(* IEC 61131-3 sources: SmartHomeNew/ (part 5) *)

(* ---- FB_Heating_Adaptive_Target.st ---- *)
// ==============================================================================
// Adaptive target calculation for heating supply temperature
// ==============================================================================
FUNCTION_BLOCK FB_Heating_Adaptive_Target
VAR_INPUT
    VI_Base_Target_Supply_Temp : REAL;
    VI_Global_Target_Temperature : REAL;
END_VAR

VAR_IN_OUT
    VI_Zone_Configs : ARRAY[1..GVL_CONSTANTS.C_MAX_HEATING_CIRCUITS] OF ST_FloorHeating_Circuit_Config;
    VI_Floor_Temps : ARRAY[1..GVL_CONSTANTS.C_MAX_HEATING_CIRCUITS] OF REAL;
    VI_Room_Temps : ARRAY[1..GVL_CONSTANTS.C_MAX_ZONES] OF REAL;
END_VAR

VAR_OUTPUT
    VO_Target_Supply_Temp : REAL;
    VO_Adaptive_Correction : REAL;
    VO_Adaptive_Effective_Delta : REAL;
    VO_Adaptive_Max_Delta : REAL;
END_VAR

VAR
    L_Adaptive_Zone_i : INT;
    L_Zone_Index : INT;
    L_Adaptive_Delta : REAL;
    L_Adaptive_Weighted_Sum : REAL;
    L_Adaptive_Weight_Total : REAL;
    L_Adaptive_Weight : REAL;
END_VAR

VO_Target_Supply_Temp := VI_Base_Target_Supply_Temp;
VO_Adaptive_Max_Delta := 0.0;
L_Adaptive_Weighted_Sum := 0.0;
L_Adaptive_Weight_Total := 0.0;
VO_Adaptive_Effective_Delta := 0.0;
VO_Adaptive_Correction := 0.0;

IF VI_Global_Target_Temperature > 0.0 THEN
    VO_Target_Supply_Temp := VI_Global_Target_Temperature;
END_IF;

FOR L_Adaptive_Zone_i := 1 TO GVL_CONSTANTS.C_MAX_HEATING_CIRCUITS DO
    L_Zone_Index := VI_Zone_Configs[L_Adaptive_Zone_i].zone;

    IF (L_Zone_Index >= 1) AND (L_Zone_Index <= GVL_CONSTANTS.C_MAX_ZONES) THEN
        CASE VI_Zone_Configs[L_Adaptive_Zone_i].control_type OF
            0:
                L_Adaptive_Delta :=
                    VI_Zone_Configs[L_Adaptive_Zone_i].design_temp -
                    VI_Floor_Temps[L_Adaptive_Zone_i];
                L_Adaptive_Weight := 0.6;
            1, 2:
                L_Adaptive_Delta :=
                    VI_Zone_Configs[L_Adaptive_Zone_i].design_temp -
                    VI_Room_Temps[L_Zone_Index];
                L_Adaptive_Weight := 1.0;
            ELSE
                L_Adaptive_Delta :=
                    VI_Zone_Configs[L_Adaptive_Zone_i].design_temp -
                    VI_Room_Temps[L_Zone_Index];
                L_Adaptive_Weight := 0.8;
        END_CASE;

        IF L_Zone_Index <= 4 THEN
            L_Adaptive_Weight := L_Adaptive_Weight * 1.2;
        ELSIF L_Zone_Index >= 9 THEN
            L_Adaptive_Weight := L_Adaptive_Weight * 0.7;
        END_IF;

        IF L_Adaptive_Weight > 2.0 THEN
            L_Adaptive_Weight := 2.0;
        ELSIF L_Adaptive_Weight < 0.2 THEN
            L_Adaptive_Weight := 0.2;
        END_IF;

        IF L_Adaptive_Delta > VO_Adaptive_Max_Delta THEN
            VO_Adaptive_Max_Delta := L_Adaptive_Delta;
        END_IF;

        L_Adaptive_Weighted_Sum := L_Adaptive_Weighted_Sum + (L_Adaptive_Delta * L_Adaptive_Weight);
        L_Adaptive_Weight_Total := L_Adaptive_Weight_Total + L_Adaptive_Weight;
    END_IF;
END_FOR;

IF L_Adaptive_Weight_Total > 0.0 THEN
    VO_Adaptive_Effective_Delta := L_Adaptive_Weighted_Sum / L_Adaptive_Weight_Total;
END_IF;

IF VO_Adaptive_Effective_Delta > 1.5 THEN
    VO_Adaptive_Correction := 2.0;
ELSIF VO_Adaptive_Effective_Delta > 0.7 THEN
    VO_Adaptive_Correction := 1.0;
ELSIF VO_Adaptive_Effective_Delta < -1.5 THEN
    VO_Adaptive_Correction := -2.0;
ELSIF VO_Adaptive_Effective_Delta < -0.7 THEN
    VO_Adaptive_Correction := -1.0;
ELSE
    VO_Adaptive_Correction := 0.0;
END_IF;

IF VO_Adaptive_Max_Delta > 2.5 AND VO_Adaptive_Correction < 2.0 THEN
    VO_Adaptive_Correction := 2.0;
END_IF;

VO_Target_Supply_Temp := VO_Target_Supply_Temp + VO_Adaptive_Correction;

IF VO_Target_Supply_Temp < 20.0 THEN
    VO_Target_Supply_Temp := 20.0;
ELSIF VO_Target_Supply_Temp > 45.0 THEN
    VO_Target_Supply_Temp := 45.0;
END_IF;

// >>> BULK_SYNC_ANCHOR: FB_Heating_Adaptive_Target <<<

(* ---- FB_Heating_Allocation_Filter.st ---- *)
// ==============================================================================
// Heating allocation filter
// Bounded policy filter between demand map and manifold control.
//
// Purpose:
// - preserve current runtime ownership;
// - avoid reconnecting legacy orchestration wrappers;
// - provide a safe insertion point for selective thermal allocation logic;
// - keep default behavior transparent when disabled.
//
// This FB does NOT own:
// - heating orchestration;
// - boiler control;
// - valve control;
// - pump control;
// - safety state;
// - output projection.
//
// Migration source:
// - useful bounded logic from FB_Heating_Thermal_Allocation;
// - useful bounded logic from FB_Heating_Decision_Context.
//
// Explicitly not migrated:
// - FB_Heating_Orchestration wrapper;
// - FB_Heating_Execution_Core wrapper;
// - FB_Heating_Override_Layer hard output authority.
// ==============================================================================
FUNCTION_BLOCK FB_Heating_Allocation_Filter
VAR_INPUT
    // Master switch for any filtering.
    // FALSE means strict passthrough: output demand equals input demand.
    VI_Enable : BOOL;

    // Enables optional priority/budget allocation.
    // FALSE means only safe availability filtering may run when VI_Enable is TRUE.
    VI_Enable_Policy_Allocation : BOOL := FALSE;

    // Current demand from FB_Heating_Demand_Map.
    VI_Manifold_Demand_Map : ARRAY[1..GVL_CONSTANTS.C_MAX_MANIFOLDS] OF BOOL;

    // Availability must come from current active owners / diagnostics.
    // TRUE means the manifold is allowed to receive demand.
    VI_Manifold_Available : ARRAY[1..GVL_CONSTANTS.C_MAX_MANIFOLDS] OF BOOL;

    // Optional policy inputs staged for future activation.
    // They intentionally stay outside existing DUT/GVL contract for now.
    VI_Manifold_Base_Priority : ARRAY[1..GVL_CONSTANTS.C_MAX_MANIFOLDS] OF INT;
    VI_Manifold_Thermal_Weight : ARRAY[1..GVL_CONSTANTS.C_MAX_MANIFOLDS] OF REAL;
    VI_Max_Thermal_Budget : REAL := REAL#0.0;
END_VAR
VAR_OUTPUT
    // Demand forwarded to FB_Heating_Manifold_Control.
    VO_Manifold_Demand_Filtered : ARRAY[1..GVL_CONSTANTS.C_MAX_MANIFOLDS] OF BOOL;

    // TRUE when at least one demanded manifold was blocked by availability or policy.
    VO_Allocation_Degraded : BOOL;

    // Diagnostic outputs for later observation/HMI integration.
    VO_Manifold_Allowed : ARRAY[1..GVL_CONSTANTS.C_MAX_MANIFOLDS] OF BOOL;
    VO_Manifold_Priority_Effective : ARRAY[1..GVL_CONSTANTS.C_MAX_MANIFOLDS] OF INT;
    VO_Thermal_Budget_Used : REAL;
END_VAR
VAR
    L_i : INT;
    L_CurrentPriority : INT;
    L_MaxPriority : INT;
    L_Used : REAL;
    L_Weight : REAL;
END_VAR

// ======================================================
// DEFAULT / TRANSPARENT MODE
// ======================================================
VO_Allocation_Degraded := FALSE;
VO_Thermal_Budget_Used := REAL#0.0;

FOR L_i := 1 TO GVL_CONSTANTS.C_MAX_MANIFOLDS DO
    VO_Manifold_Demand_Filtered[L_i] := VI_Manifold_Demand_Map[L_i];
    VO_Manifold_Allowed[L_i] := TRUE;
    VO_Manifold_Priority_Effective[L_i] := VI_Manifold_Base_Priority[L_i];
END_FOR;

IF NOT VI_Enable THEN
    RETURN;
END_IF;

// ======================================================
// SAFE AVAILABILITY FILTER
// ======================================================
FOR L_i := 1 TO GVL_CONSTANTS.C_MAX_MANIFOLDS DO
    VO_Manifold_Allowed[L_i] := VI_Manifold_Available[L_i];

    IF VI_Manifold_Demand_Map[L_i] AND NOT VO_Manifold_Allowed[L_i] THEN
        VO_Manifold_Demand_Filtered[L_i] := FALSE;
        VO_Allocation_Degraded := TRUE;
    END_IF;
END_FOR;

// ======================================================
// OPTIONAL POLICY / THERMAL BUDGET ALLOCATION
// ======================================================
IF NOT VI_Enable_Policy_Allocation THEN
    RETURN;
END_IF;

// Invalid or unset budget means do not apply budget shedding.
IF VI_Max_Thermal_Budget <= REAL#0.0 THEN
    RETURN;
END_IF;

// Clear filtered demand before rebuilding it by priority and budget.
FOR L_i := 1 TO GVL_CONSTANTS.C_MAX_MANIFOLDS DO
    VO_Manifold_Demand_Filtered[L_i] := FALSE;
END_FOR;

// Find max priority among demanded and allowed manifolds.
L_MaxPriority := 0;
FOR L_i := 1 TO GVL_CONSTANTS.C_MAX_MANIFOLDS DO
    IF VI_Manifold_Demand_Map[L_i] AND VO_Manifold_Allowed[L_i] THEN
        IF VO_Manifold_Priority_Effective[L_i] > L_MaxPriority THEN
            L_MaxPriority := VO_Manifold_Priority_Effective[L_i];
        END_IF;
    END_IF;
END_FOR;

L_Used := REAL#0.0;

FOR L_CurrentPriority := L_MaxPriority TO 0 BY -1 DO
    FOR L_i := 1 TO GVL_CONSTANTS.C_MAX_MANIFOLDS DO
        IF VI_Manifold_Demand_Map[L_i]
           AND VO_Manifold_Allowed[L_i]
           AND (VO_Manifold_Priority_Effective[L_i] = L_CurrentPriority) THEN

            L_Weight := VI_Manifold_Thermal_Weight[L_i];
            IF L_Weight <= REAL#0.0 THEN
                L_Weight := REAL#1.0;
            END_IF;

            IF (L_Used + L_Weight) <= VI_Max_Thermal_Budget THEN
                VO_Manifold_Demand_Filtered[L_i] := TRUE;
                L_Used := L_Used + L_Weight;
            ELSE
                VO_Allocation_Degraded := TRUE;
            END_IF;
        END_IF;
    END_FOR;
END_FOR;

VO_Thermal_Budget_Used := L_Used;

END_FUNCTION_BLOCK
// >>> BULK_SYNC_ANCHOR: FB_Heating_Allocation_Filter <<<

(* ---- FB_Heating_Boiler_Control.st ---- *)
// ==============================================================================
// Heating boiler control helper
// ==============================================================================
FUNCTION_BLOCK FB_Heating_Boiler_Control
VAR_INPUT
    VI_System_Time_MS : UDINT;
    VI_IsActivePLC : BOOL;
    VI_DHW_Heating_Demand : BOOL;
    VI_DHW_Target_Temp : REAL;
    VI_Target_Supply_Temp : REAL;
    VI_Freeze_Mode_Active : BOOL;
    VI_Policy_Degraded : BOOL;
    VI_Manifold_Pumps : ARRAY[1..GVL_CONSTANTS.C_MAX_MANIFOLDS] OF BOOL;
    VI_Manifold_Valves : ARRAY[1..GVL_CONSTANTS.C_MAX_MANIFOLDS] OF REAL;
    VI_Boiler_Flame_Status : ARRAY[1..GVL_CONSTANTS.C_MAX_BOILERS] OF BOOL;
    VI_Boiler_Error_Status : ARRAY[1..GVL_CONSTANTS.C_MAX_BOILERS] OF BOOL;
    VI_Boiler_OT_Online : ARRAY[1..GVL_CONSTANTS.C_MAX_BOILERS] OF BOOL;
END_VAR
VAR_IN_OUT
    VI_Boiler_Modulation : ARRAY[1..GVL_CONSTANTS.C_MAX_BOILERS] OF REAL;
END_VAR
VAR_OUTPUT
    VO_Boiler_OT_Enable : ARRAY[1..GVL_CONSTANTS.C_MAX_BOILERS] OF BOOL;
    VO_Boiler_OT_Setpoint : ARRAY[1..GVL_CONSTANTS.C_MAX_BOILERS] OF REAL;
    VO_Boiler_Status : ARRAY[1..GVL_CONSTANTS.C_MAX_BOILERS] OF ST_Boiler_Status;
    VO_Any_Subsystem_Degraded : BOOL;
    VO_Lead_Boiler : BYTE;
    VO_Demand_Power : REAL;
END_VAR
VAR
    L_i : INT;
    L_Delta_MS : UDINT;
    L_Last_Scan_Time : UDINT;
    L_Scan_Time_Init : BOOL := FALSE;
    L_Boiler_Request_Enable : ARRAY[1..GVL_CONSTANTS.C_MAX_BOILERS] OF BOOL;
    L_Boiler_Request_Setpoint : ARRAY[1..GVL_CONSTANTS.C_MAX_BOILERS] OF REAL;
    L_Boiler_OT_Command_Valid : ARRAY[1..GVL_CONSTANTS.C_MAX_BOILERS] OF BOOL;
    L_Transport_Degraded : BOOL;
    L_Available_Count : UINT;
    L_Active_Count : UINT;
    L_Any_Transport_Degraded : BOOL;
    L_Any_Ignition_Timeout : BOOL;
    L_Any_Flame : BOOL;
    L_Empty_Boiler_Status : ST_Boiler_Status;
    L_Boiler_Life : ARRAY[1..GVL_CONSTANTS.C_MAX_BOILERS] OF FB_Lifetime_Predictor;
    fbBoilerCascade : FB_Boiler_Cascade_Manager;
    fbBoilerOpenTherm : FB_Boiler_OpenTherm_Interface;
END_VAR

VO_Any_Subsystem_Degraded := FALSE;
VO_Lead_Boiler := 0;
VO_Demand_Power := 0.0;

L_Available_Count := 0;
L_Active_Count := 0;
L_Any_Transport_Degraded := FALSE;
L_Any_Ignition_Timeout := FALSE;
L_Any_Flame := FALSE;

FOR L_i := 1 TO GVL_CONSTANTS.C_MAX_BOILERS DO
    L_Boiler_Request_Enable[L_i] := FALSE;
    L_Boiler_Request_Setpoint[L_i] := 0.0;
    L_Boiler_OT_Command_Valid[L_i] := FALSE;
    VO_Boiler_OT_Enable[L_i] := FALSE;
    VO_Boiler_OT_Setpoint[L_i] := 0.0;
    VO_Boiler_Status[L_i] := L_Empty_Boiler_Status;
END_FOR;

FOR L_i := 1 TO GVL_CONSTANTS.C_MAX_MANIFOLDS DO
    IF VI_Manifold_Pumps[L_i] THEN
        VO_Demand_Power := VO_Demand_Power + VI_Manifold_Valves[L_i];
    END_IF;
END_FOR;

IF VI_Freeze_Mode_Active AND VO_Demand_Power < 20.0 THEN
    VO_Demand_Power := 20.0;
END_IF;

IF VI_Policy_Degraded THEN
    IF VO_Demand_Power > 60.0 THEN
        VO_Demand_Power := 60.0;
    END_IF;
END_IF;

fbBoilerCascade(
    VI_Enable := VI_IsActivePLC AND ((VO_Demand_Power > GVL_CONSTANTS.C_BOILER_CASCADE_MIN_DEMAND) OR VI_Freeze_Mode_Active OR VI_DHW_Heating_Demand),
    VI_System_Time_MS := VI_System_Time_MS,
    VI_Boiler_Stop := FALSE,
    VI_DHW_Heating_Demand := VI_DHW_Heating_Demand,
    VI_DHW_Target_Temp := VI_DHW_Target_Temp,
    VI_Target_Supply_Temp := VI_Target_Supply_Temp,
    VI_Demand_Power := VO_Demand_Power,
    VI_Boiler_Flame_Status := VI_Boiler_Flame_Status,
    VI_Boiler_Error_Status := VI_Boiler_Error_Status,
    VI_Boiler_OT_Online := VI_Boiler_OT_Online,
    VI_Boiler_Modulation := VI_Boiler_Modulation,
    VO_Boiler_Enable => L_Boiler_Request_Enable,
    VO_Boiler_Setpoint => L_Boiler_Request_Setpoint,
    VO_Lead_Boiler => VO_Lead_Boiler
);

FOR L_i := 1 TO GVL_CONSTANTS.C_MAX_BOILERS DO
    IF L_Boiler_Request_Enable[L_i] THEN
        L_Boiler_Request_Setpoint[L_i] := LIMIT(
            GVL_CONSTANTS.C_BOILER_SETPOINT_MIN,
            L_Boiler_Request_Setpoint[L_i],
            80.0
        );
    END_IF;
END_FOR;

FOR L_i := 1 TO GVL_CONSTANTS.C_MAX_BOILERS DO
    IF NOT VI_Boiler_OT_Online[L_i] OR VI_Boiler_Error_Status[L_i] THEN
        L_Boiler_Request_Enable[L_i] := FALSE;
        L_Boiler_Request_Setpoint[L_i] := 0.0;
    END_IF;
END_FOR;

fbBoilerOpenTherm(
    VI_Enable := L_Boiler_Request_Enable,
    VI_Setpoint := L_Boiler_Request_Setpoint,
    VI_OT_Online := VI_Boiler_OT_Online,
    VI_OT_Error := VI_Boiler_Error_Status,
    VO_OT_Enable => VO_Boiler_OT_Enable,
    VO_OT_Setpoint => VO_Boiler_OT_Setpoint,
    VO_OT_Command_Valid => L_Boiler_OT_Command_Valid
);

FOR L_i := 1 TO GVL_CONSTANTS.C_MAX_BOILERS DO

    L_Transport_Degraded :=
        L_Boiler_Request_Enable[L_i] AND
        (
            NOT L_Boiler_OT_Command_Valid[L_i] OR
            NOT VI_Boiler_OT_Online[L_i] OR
            VI_Boiler_Error_Status[L_i]
        );

    VO_Boiler_Status[L_i].OT_Online := VI_Boiler_OT_Online[L_i];
    VO_Boiler_Status[L_i].OT_Command_Valid := L_Boiler_OT_Command_Valid[L_i];
    VO_Boiler_Status[L_i].OT_Transport_Degraded := L_Transport_Degraded;
    VO_Boiler_Status[L_i].OT_Adapter_Error :=
        GVL_OPENTHERM_ADAPTER.G_Status[L_i].Adapter_Error;

    VO_Boiler_Status[L_i].Active := L_Boiler_Request_Enable[L_i];
    VO_Boiler_Status[L_i].Running := VI_Boiler_Flame_Status[L_i];
    VO_Boiler_Status[L_i].Warning := L_Transport_Degraded;
    VO_Boiler_Status[L_i].Error := VI_Boiler_Error_Status[L_i];

    VO_Boiler_Status[L_i].Available :=
        VI_Boiler_OT_Online[L_i] AND
        NOT VI_Boiler_Error_Status[L_i] AND
        NOT L_Transport_Degraded;

    VO_Boiler_Status[L_i].Selected_By_Cascade :=
        L_Boiler_Request_Enable[L_i];

    VO_Boiler_Status[L_i].Transport_Missing :=
        NOT VI_Boiler_OT_Online[L_i];

    VO_Boiler_Status[L_i].Flame_Missing :=
        L_Boiler_Request_Enable[L_i] AND
        NOT VI_Boiler_Flame_Status[L_i] AND
        NOT L_Transport_Degraded;

    VO_Boiler_Status[L_i].Ignition_Timeout :=
        VO_Boiler_Status[L_i].Flame_Missing AND
        (GVL_STATE.G_Boiler_OT_Command_Age_MS[L_i] > 30000);

    VO_Boiler_Status[L_i].Degraded :=
        L_Transport_Degraded OR
        VO_Boiler_Status[L_i].Ignition_Timeout;

    // ======================================================
    // CASCADE AGGREGATION
    // ======================================================
    IF VO_Boiler_Status[L_i].Available THEN
        L_Available_Count := L_Available_Count + 1;
    END_IF;

    IF VO_Boiler_Status[L_i].Selected_By_Cascade THEN
        L_Active_Count := L_Active_Count + 1;
    END_IF;

    IF VI_Boiler_Flame_Status[L_i] THEN
        L_Any_Flame := TRUE;
    END_IF;

    IF L_Transport_Degraded THEN
        L_Any_Transport_Degraded := TRUE;
    END_IF;

    IF VO_Boiler_Status[L_i].Ignition_Timeout THEN
        L_Any_Ignition_Timeout := TRUE;
    END_IF;

    IF VO_Boiler_Status[L_i].Degraded THEN
        VO_Any_Subsystem_Degraded := TRUE;
    END_IF;

END_FOR;

// ======================================================
// GLOBAL CASCADE SEMANTIC STATE
// ======================================================
GVL_STATE.G_Heating_Cascade_Active_Boilers := L_Active_Count;
GVL_STATE.G_Heating_Cascade_Available_Boilers := L_Available_Count;

GVL_STATE.G_Heating_Cascade_Available :=
    (L_Available_Count > 0);

GVL_STATE.G_Heating_Cascade_Partial_Capacity :=
    (L_Available_Count > 0) AND
    (L_Available_Count < GVL_CONSTANTS.C_MAX_BOILERS);

GVL_STATE.G_Heating_Cascade_Transport_Degraded :=
    L_Any_Transport_Degraded;

GVL_STATE.G_Heating_Cascade_Ignition_Timeout :=
    L_Any_Ignition_Timeout;

GVL_STATE.G_Heating_Cascade_No_Flame :=
    (L_Active_Count > 0) AND
    NOT L_Any_Flame;

GVL_STATE.G_Heating_Cascade_Degraded :=
    GVL_STATE.G_Heating_Cascade_Transport_Degraded OR
    GVL_STATE.G_Heating_Cascade_Ignition_Timeout OR
    GVL_STATE.G_Heating_Cascade_Partial_Capacity;

END_FUNCTION_BLOCK

(* ---- FB_Heating_Circuit_Control.st ---- *)
// ==============================================================================
// Heating circuit control helper
//
// Internal refactoring helper for FB_Heating_System_Manager.
// Owns per-circuit sensor validation, temperature source fallback,
// floor-heating controller call, overheat shutdown, and rule action projection.
//
// Temperature source selection is confidence-aware:
// - range invalid still blocks that source;
// - passive input-quality confidence can prefer a healthier fallback;
// - degraded-but-range-valid sources remain operational if no better source exists.
// ==============================================================================
FUNCTION_BLOCK FB_Heating_Circuit_Control
VAR_INPUT
    VI_System_Time_MS : UDINT;
    VI_Current_Hour : UINT;
    VI_IsActivePLC : BOOL;
    VI_Config : ST_Heating_Config;
    VI_Tariff : ST_Tariff_Config;
    VI_Scenario_Adjust : REAL;
END_VAR

VAR_IN_OUT
    VI_Zone_Configs : ARRAY[1..GVL_CONSTANTS.C_MAX_HEATING_CIRCUITS] OF ST_FloorHeating_Circuit_Config;
    VI_Floor_Temps : ARRAY[1..GVL_CONSTANTS.C_MAX_HEATING_CIRCUITS] OF REAL;
    VI_Room_Temps : ARRAY[1..16] OF REAL;
    VI_Rule_Actions : ARRAY[1..GVL_CONSTANTS.C_MAX_RULES] OF ST_Rule_Action;
END_VAR

VAR_OUTPUT
    VO_Zone_Valves : ARRAY[1..GVL_CONSTANTS.C_MAX_HEATING_CIRCUITS] OF BOOL;
    VO_Heating_Sensor_Fault : BOOL;
END_VAR

VAR
    L_i : INT;
    L_j : INT;
    L_Climate_Zone_ID : INT;
    L_Zone_Config : ST_FloorHeating_Circuit_Config;
    L_Current_Temp : REAL;
    L_Sensor_Error : BOOL;
    L_Floor_Source_Valid : BOOL;
    L_Room_Source_Valid : BOOL;
    L_Floor_Confidence : REAL;
    L_Room_Confidence : REAL;
    L_Min_Source_Confidence : REAL;

    L_Floor_Controllers : ARRAY[1..GVL_CONSTANTS.C_MAX_HEATING_CIRCUITS] OF FB_FloorHeating_Controller;
    L_Overheat_Timer : ARRAY[1..GVL_CONSTANTS.C_MAX_HEATING_CIRCUITS] OF FB_System_Timer;
    fbFloorTempValidator : ARRAY[1..GVL_CONSTANTS.C_MAX_HEATING_CIRCUITS] OF FB_Analog_Validator;
    fbRoomTempValidator : ARRAY[1..16] OF FB_Analog_Validator;
END_VAR

VO_Heating_Sensor_Fault := FALSE;
L_Min_Source_Confidence := GVL_INPUT_VALIDATION_CONFIG.G_Min_Sensor_Confidence;

FOR L_i := 1 TO GVL_CONSTANTS.C_MAX_HEATING_CIRCUITS DO
    fbFloorTempValidator[L_i](
        VI_Value := VI_Floor_Temps[L_i],
        VI_Min_Valid := -40.0,
        VI_Max_Valid := 120.0,
        VI_Fallback_Mode := 0
    );

    L_Climate_Zone_ID := VI_Zone_Configs[L_i].zone;
    IF L_Climate_Zone_ID >= 1 AND L_Climate_Zone_ID <= 16 THEN
        fbRoomTempValidator[L_Climate_Zone_ID](
            VI_Value := VI_Room_Temps[L_Climate_Zone_ID],
            VI_Min_Valid := -40.0,
            VI_Max_Valid := 120.0,
            VI_Fallback_Mode := 0
        );
    END_IF;

    L_Floor_Source_Valid := NOT fbFloorTempValidator[L_i].VO_Error;
    L_Room_Source_Valid :=
        (L_Climate_Zone_ID >= 1) AND
        (L_Climate_Zone_ID <= 16) AND
        (NOT fbRoomTempValidator[L_Climate_Zone_ID].VO_Error);

    L_Floor_Confidence := REAL#1.0;
    IF GVL_INPUT_QUALITY.G_Floor_Temp_Quality[L_i].Quality_Visible THEN
        L_Floor_Confidence := GVL_INPUT_QUALITY.G_Floor_Temp_Quality[L_i].Confidence;
    END_IF;

    L_Room_Confidence := REAL#1.0;
    IF (L_Climate_Zone_ID >= 1) AND (L_Climate_Zone_ID <= 16) THEN
        IF GVL_INPUT_QUALITY.G_Room_Temp_Quality[L_Climate_Zone_ID].Quality_Visible THEN
            L_Room_Confidence := GVL_INPUT_QUALITY.G_Room_Temp_Quality[L_Climate_Zone_ID].Confidence;
        END_IF;
    END_IF;

    IF L_Floor_Confidence < REAL#0.0 THEN
        L_Floor_Confidence := REAL#0.0;
    ELSIF L_Floor_Confidence > REAL#1.0 THEN
        L_Floor_Confidence := REAL#1.0;
    END_IF;

    IF L_Room_Confidence < REAL#0.0 THEN
        L_Room_Confidence := REAL#0.0;
    ELSIF L_Room_Confidence > REAL#1.0 THEN
        L_Room_Confidence := REAL#1.0;
    END_IF;

    // Floor overheat protection remains floor-bound and range-validity based.
    L_Overheat_Timer[L_i](
        IN := L_Floor_Source_Valid AND (fbFloorTempValidator[L_i].VO_Value > VI_Config.Overheat_Threshold),
        PT := T#60s,
        VI_System_Time_MS := VI_System_Time_MS
    );

    L_Current_Temp := REAL#0.0;
    L_Sensor_Error := FALSE;

    IF VI_Zone_Configs[L_i].control_type = 1 OR VI_Zone_Configs[L_i].control_type = 2 THEN
        // Primary: room air temperature. If room quality is degraded and floor
        // source is healthier, prefer floor fallback without declaring hard fault.
        IF L_Room_Source_Valid AND
           ((L_Room_Confidence >= L_Min_Source_Confidence) OR NOT L_Floor_Source_Valid OR (L_Room_Confidence >= L_Floor_Confidence)) THEN
            L_Current_Temp := fbRoomTempValidator[L_Climate_Zone_ID].VO_Value;
        ELSIF L_Floor_Source_Valid THEN
            L_Current_Temp := fbFloorTempValidator[L_i].VO_Value;
        ELSIF L_Room_Source_Valid THEN
            L_Current_Temp := fbRoomTempValidator[L_Climate_Zone_ID].VO_Value;
        ELSE
            L_Sensor_Error := TRUE;
        END_IF;
    ELSE
        // Primary: floor temperature. If floor quality is degraded and room
        // source is healthier, prefer room fallback without declaring hard fault.
        IF L_Floor_Source_Valid AND
           ((L_Floor_Confidence >= L_Min_Source_Confidence) OR NOT L_Room_Source_Valid OR (L_Floor_Confidence >= L_Room_Confidence)) THEN
            L_Current_Temp := fbFloorTempValidator[L_i].VO_Value;
        ELSIF L_Room_Source_Valid THEN
            L_Current_Temp := fbRoomTempValidator[L_Climate_Zone_ID].VO_Value;
        ELSIF L_Floor_Source_Valid THEN
            L_Current_Temp := fbFloorTempValidator[L_i].VO_Value;
        ELSE
            L_Sensor_Error := TRUE;
        END_IF;
    END_IF;

    IF L_Sensor_Error THEN
        VO_Heating_Sensor_Fault := TRUE;
        VO_Zone_Valves[L_i] := FALSE;
    ELSE
        L_Zone_Config := VI_Zone_Configs[L_i];
        L_Zone_Config.design_temp := L_Zone_Config.design_temp + VI_Scenario_Adjust;

        L_Floor_Controllers[L_i](
            VI_Current_Temp := L_Current_Temp,
            VI_Config := L_Zone_Config,
            VI_Tariff := VI_Tariff,
            VI_Current_Hour := VI_Current_Hour,
            VI_IsActivePLC := VI_IsActivePLC,
            VI_System_Time_MS := VI_System_Time_MS,
            VO_Valve_Bool => VO_Zone_Valves[L_i]
        );
    END_IF;

    IF L_Overheat_Timer[L_i].Q THEN
        VO_Zone_Valves[L_i] := FALSE;
    END_IF;

    FOR L_j := 1 TO GVL_CONSTANTS.C_MAX_RULES DO
        IF VI_Rule_Actions[L_j].Active AND VI_Rule_Actions[L_j].Target_ID = L_i THEN
            IF VI_Rule_Actions[L_j].Action_Type = E_Rule_Action_Type.ACTION_SET_FLOOR_HEATING THEN
                VO_Zone_Valves[L_i] := (VI_Rule_Actions[L_j].Value > REAL#0.5);
            END_IF;
        END_IF;
    END_FOR;
END_FOR;

// >>> BULK_SYNC_ANCHOR: FB_Heating_Circuit_Control <<<
END_FUNCTION_BLOCK

(* ---- FB_Heating_Circuit_Explainability_Adapter.st ---- *)
// ==============================================================================
// Heating circuit explainability adapter
//
// Projection-to-explainability adapter.
//
// DOES NOT own runtime authority.
// DOES NOT own outputs.
// DOES NOT close valves.
// DOES NOT modify heating demand.
// DOES NOT override runtime decisions.
//
// Reads canonical runtime projection contracts and publishes legacy-compatible
// circuit explainability surfaces for HMI/diagnostics/supervisory visibility.
// ==============================================================================
FUNCTION_BLOCK FB_Heating_Circuit_Explainability_Adapter
VAR_INPUT
    VI_Enable : BOOL;
END_VAR

VAR
    L_i : INT;
END_VAR

IF NOT VI_Enable THEN
    RETURN;
END_IF;

FOR L_i := 1 TO GVL_CONSTANTS.C_MAX_HEATING_CIRCUITS DO
    GVL_Heating_Circuit_Explainability.G_Source_Selection_Visible[L_i] :=
        GVL_Heating_Runtime_Projection.G_Circuit_Projection[L_i].Visible;

    GVL_Heating_Circuit_Explainability.G_Selected_Source_Code[L_i] :=
        GVL_Heating_Runtime_Projection.G_Circuit_Projection[L_i].Selected_Source_Code;

    CASE GVL_Heating_Runtime_Projection.G_Circuit_Projection[L_i].Selected_Source_Code OF
        1:
            GVL_Heating_Circuit_Explainability.G_Selected_Source_Text[L_i] := 'room';
        2:
            GVL_Heating_Circuit_Explainability.G_Selected_Source_Text[L_i] := 'floor';
    ELSE
        GVL_Heating_Circuit_Explainability.G_Selected_Source_Text[L_i] := 'none';
    END_CASE;

    GVL_Heating_Circuit_Explainability.G_Fallback_Active[L_i] :=
        GVL_Heating_Runtime_Projection.G_Circuit_Projection[L_i].Fallback_Active;

    GVL_Heating_Circuit_Explainability.G_Source_Degraded[L_i] :=
        GVL_Heating_Runtime_Projection.G_Circuit_Projection[L_i].Source_Degraded;

    GVL_Heating_Circuit_Explainability.G_Selected_Source_Confidence[L_i] :=
        GVL_Heating_Runtime_Projection.G_Circuit_Projection[L_i].Selected_Source_Confidence;

    // Primary/fallback confidence remain legacy-compatible fields. The runtime
    // projection intentionally exposes selected confidence only, so these fields
    // mirror the selected source confidence until a dedicated richer projection
    // contract is introduced.
    GVL_Heating_Circuit_Explainability.G_Primary_Source_Confidence[L_i] :=
        GVL_Heating_Runtime_Projection.G_Circuit_Projection[L_i].Selected_Source_Confidence;

    GVL_Heating_Circuit_Explainability.G_Fallback_Source_Confidence[L_i] :=
        GVL_Heating_Runtime_Projection.G_Circuit_Projection[L_i].Selected_Source_Confidence;

    GVL_Heating_Circuit_Explainability.G_Reason_Code[L_i] :=
        GVL_Heating_Runtime_Projection.G_Circuit_Projection[L_i].Reason_Code;

    GVL_Heating_Circuit_Explainability.G_Reason_Text[L_i] :=
        GVL_Heating_Runtime_Projection.G_Circuit_Projection[L_i].Reason_Text;

    GVL_Heating_Circuit_Explainability.G_Source_Switched_Event[L_i] :=
        GVL_Heating_Runtime_Projection.G_Circuit_Projection[L_i].Source_Switched_Event;

    GVL_Heating_Circuit_Explainability.G_Fallback_Activated_Event[L_i] :=
        GVL_Heating_Runtime_Projection.G_Circuit_Projection[L_i].Fallback_Activated_Event;

    GVL_Heating_Circuit_Explainability.G_Fallback_Recovered_Event[L_i] :=
        GVL_Heating_Runtime_Projection.G_Circuit_Projection[L_i].Fallback_Recovered_Event;

    GVL_Heating_Circuit_Explainability.G_Source_Loss_Event[L_i] :=
        GVL_Heating_Runtime_Projection.G_Circuit_Projection[L_i].Source_Loss_Event;

    GVL_Heating_Circuit_Explainability.G_Last_Event_MS[L_i] :=
        GVL_Heating_Runtime_Projection.G_Circuit_Projection[L_i].Last_Event_MS;

    GVL_Heating_Circuit_Explainability.G_Last_Event_Code[L_i] :=
        GVL_Heating_Runtime_Projection.G_Circuit_Projection[L_i].Last_Event_Code;

    GVL_Heating_Circuit_Explainability.G_Last_Event_Text[L_i] :=
        GVL_Heating_Runtime_Projection.G_Circuit_Projection[L_i].Last_Event_Text;
END_FOR;

END_FUNCTION_BLOCK
// >>> BULK_SYNC_ANCHOR: FB_Heating_Circuit_Explainability_Adapter <<<

(* ---- FB_Heating_Decision_Context.st ---- *)
FUNCTION_BLOCK FB_Heating_Decision_Context
VAR_INPUT
    VI_Manifold_Pump_In_Service : ARRAY[1..GVL_CONSTANTS.C_MAX_MANIFOLDS] OF BOOL;
    VI_Manifold_Pressure_Fault : ARRAY[1..GVL_CONSTANTS.C_MAX_MANIFOLDS] OF BOOL;
    VI_Manifold_Current_Fault : ARRAY[1..GVL_CONSTANTS.C_MAX_MANIFOLDS] OF BOOL;
    VI_Manifold_Thermal_Weight : ARRAY[1..GVL_CONSTANTS.C_MAX_MANIFOLDS] OF REAL;
    VI_Manifold_Priority : ARRAY[1..GVL_CONSTANTS.C_MAX_MANIFOLDS] OF INT;
    VI_Max_Thermal_Budget : REAL;
END_VAR
VAR_OUTPUT
    VO_Manifold_Allowed : ARRAY[1..GVL_CONSTANTS.C_MAX_MANIFOLDS] OF BOOL;
    VO_Manifold_Enabled : ARRAY[1..GVL_CONSTANTS.C_MAX_MANIFOLDS] OF BOOL;
    VO_Heating_Degraded : BOOL;
END_VAR
VAR
    L_i : INT;
    L_j : INT;
    L_Used : REAL;
    L_Selected : ARRAY[1..GVL_CONSTANTS.C_MAX_MANIFOLDS] OF BOOL;
    L_MaxPriority : INT;
    L_CurrentPriority : INT;
END_VAR

VO_Heating_Degraded := FALSE;

// STEP 1: Allowed
FOR L_i := 1 TO GVL_CONSTANTS.C_MAX_MANIFOLDS DO
    VO_Manifold_Allowed[L_i] := TRUE;

    IF NOT VI_Manifold_Pump_In_Service[L_i] THEN
        VO_Manifold_Allowed[L_i] := FALSE;
    END_IF;

    IF VI_Manifold_Pressure_Fault[L_i] THEN
        VO_Manifold_Allowed[L_i] := FALSE;
    END_IF;

    IF VI_Manifold_Current_Fault[L_i] THEN
        VO_Manifold_Allowed[L_i] := FALSE;
    END_IF;

    IF NOT VO_Manifold_Allowed[L_i] THEN
        VO_Heating_Degraded := TRUE;
    END_IF;
END_FOR;

// STEP 2: find max priority
L_MaxPriority := 0;
FOR L_i := 1 TO GVL_CONSTANTS.C_MAX_MANIFOLDS DO
    IF VI_Manifold_Priority[L_i] > L_MaxPriority THEN
        L_MaxPriority := VI_Manifold_Priority[L_i];
    END_IF;
END_FOR;

// STEP 3: allocation by priority + budget
FOR L_i := 1 TO GVL_CONSTANTS.C_MAX_MANIFOLDS DO
    VO_Manifold_Enabled[L_i] := FALSE;
END_FOR;

L_Used := 0.0;

FOR L_CurrentPriority := L_MaxPriority TO 1 BY -1 DO

    FOR L_i := 1 TO GVL_CONSTANTS.C_MAX_MANIFOLDS DO

        IF (VI_Manifold_Priority[L_i] = L_CurrentPriority) AND VO_Manifold_Allowed[L_i] THEN

            IF (L_Used + VI_Manifold_Thermal_Weight[L_i]) <= VI_Max_Thermal_Budget THEN
                VO_Manifold_Enabled[L_i] := TRUE;
                L_Used := L_Used + VI_Manifold_Thermal_Weight[L_i];
            END_IF;

        END_IF;

    END_FOR;

END_FOR;

(* ---- FB_Heating_Demand_Map.st ---- *)
FUNCTION_BLOCK FB_Heating_Demand_Map
VAR_INPUT
    VI_Zone_Valves : ARRAY[1..GVL_CONSTANTS.C_MAX_HEATING_CIRCUITS] OF BOOL;
    VI_Zone_Configs : ARRAY[1..GVL_CONSTANTS.C_MAX_HEATING_CIRCUITS] OF ST_FloorHeating_Circuit_Config;
END_VAR
VAR_OUTPUT
    VO_Zone_Active_Map : ARRAY[1..GVL_CONSTANTS.C_MAX_MANIFOLDS] OF BOOL;
END_VAR
VAR
    L_i : INT;
    L_Manifold_ID : INT;
END_VAR

FOR L_i := 1 TO GVL_CONSTANTS.C_MAX_MANIFOLDS DO
    VO_Zone_Active_Map[L_i] := FALSE;
END_FOR;

FOR L_i := 1 TO GVL_CONSTANTS.C_MAX_HEATING_CIRCUITS DO
    IF VI_Zone_Valves[L_i] THEN
        L_Manifold_ID := VI_Zone_Configs[L_i].manifold_id;
        IF L_Manifold_ID >= 1 AND L_Manifold_ID <= GVL_CONSTANTS.C_MAX_MANIFOLDS THEN
            VO_Zone_Active_Map[L_Manifold_ID] := TRUE;
        END_IF;
    END_IF;
END_FOR;

END_FUNCTION_BLOCK
// >>> BULK_SYNC_ANCHOR: FB_Heating_Demand_Map <<<

(* ---- FB_Heating_Diagnostics.st ---- *)
FUNCTION_BLOCK FB_Heating_Diagnostics
VAR_INPUT
    VI_System_Time_MS : UDINT;
END_VAR
VAR
    fbDiagEventManager : FB_Diagnostics_Event_Manager;
    L_i : INT;
    L_Any_Heating_Device_Failed : BOOL;
    L_Critical_Fault : BOOL;
END_VAR

// ======================================================
// DEVICE AVAILABILITY
// ======================================================
GVL_STATUS.G_Diagnostics.Backup_Pump_Out_Of_Service := NOT GVL_CONFIG.G_Backup_Circulation_Pump_In_Service;
GVL_STATUS.G_Diagnostics.Electric_Heater_Out_Of_Service := NOT GVL_CONFIG.G_Electric_Heater_In_Service;

L_Any_Heating_Device_Failed :=
    NOT GVL_CONFIG.G_Backup_Circulation_Pump_In_Service OR
    NOT GVL_CONFIG.G_Electric_Heater_In_Service;

fbDiagEventManager(
    VI_Code := GVL_CONFIG.ERR_BACKUP_PUMP_OUT_OF_SERVICE,
    VI_Severity := 2,
    VI_Active := NOT GVL_CONFIG.G_Backup_Circulation_Pump_In_Service,
    VI_Timestamp := VI_System_Time_MS,
    VI_Source := 400,
    VIO_Events := GVL_STATUS.G_Diagnostics_Events,
    VIO_Count := GVL_STATUS.G_Diagnostics_Count
);

fbDiagEventManager(
    VI_Code := GVL_CONFIG.ERR_ELECTRIC_HEATER_OUT_OF_SERVICE,
    VI_Severity := 2,
    VI_Active := NOT GVL_CONFIG.G_Electric_Heater_In_Service,
    VI_Timestamp := VI_System_Time_MS,
    VI_Source := 401,
    VIO_Events := GVL_STATUS.G_Diagnostics_Events,
    VIO_Count := GVL_STATUS.G_Diagnostics_Count
);

// ======================================================
// MANIFOLDS
// ======================================================
FOR L_i := 1 TO GVL_CONSTANTS.C_MAX_MANIFOLDS DO
    GVL_STATUS.G_Diagnostics.Manifold_Pump_Out_Of_Service[L_i] := NOT GVL_CONFIG.G_Manifold_Pump_In_Service[L_i];

    IF NOT GVL_CONFIG.G_Manifold_Pump_In_Service[L_i] THEN
        L_Any_Heating_Device_Failed := TRUE;
    END_IF;

    fbDiagEventManager(
        VI_Code := GVL_CONFIG.ERR_MANIFOLD_PUMP_OUT_OF_SERVICE,
        VI_Severity := 2,
        VI_Active := NOT GVL_CONFIG.G_Manifold_Pump_In_Service[L_i],
        VI_Timestamp := VI_System_Time_MS,
        VI_Source := 410 + L_i,
        VIO_Events := GVL_STATUS.G_Diagnostics_Events,
        VIO_Count := GVL_STATUS.G_Diagnostics_Count
    );
END_FOR;

// ======================================================
// DHW
// ======================================================
GVL_STATUS.G_Diagnostics.DHW_Heating_Pump_Out_Of_Service := NOT GVL_CONFIG.G_DHW_Heating_Pump_In_Service;
GVL_STATUS.G_Diagnostics.DHW_Circ_Pump_Out_Of_Service := NOT GVL_CONFIG.G_DHW_Circ_Pump_In_Service;

IF NOT GVL_CONFIG.G_DHW_Heating_Pump_In_Service OR
   NOT GVL_CONFIG.G_DHW_Circ_Pump_In_Service THEN
    L_Any_Heating_Device_Failed := TRUE;
END_IF;

fbDiagEventManager(
    VI_Code := GVL_CONFIG.ERR_DHW_HEATING_PUMP_OUT_OF_SERVICE,
    VI_Severity := 2,
    VI_Active := NOT GVL_CONFIG.G_DHW_Heating_Pump_In_Service,
    VI_Timestamp := VI_System_Time_MS,
    VI_Source := 420,
    VIO_Events := GVL_STATUS.G_Diagnostics_Events,
    VIO_Count := GVL_STATUS.G_Diagnostics_Count
);

fbDiagEventManager(
    VI_Code := GVL_CONFIG.ERR_DHW_CIRC_PUMP_OUT_OF_SERVICE,
    VI_Severity := 2,
    VI_Active := NOT GVL_CONFIG.G_DHW_Circ_Pump_In_Service,
    VI_Timestamp := VI_System_Time_MS,
    VI_Source := 421,
    VIO_Events := GVL_STATUS.G_Diagnostics_Events,
    VIO_Count := GVL_STATUS.G_Diagnostics_Count
);

// ======================================================
// CRITICAL FAULTS
// ======================================================
L_Critical_Fault := GVL_STATE.G_Freeze_Hardware_Failed;

fbDiagEventManager(
    VI_Code := GVL_CONFIG.ERR_FREEZE_HARDWARE_FAILED,
    VI_Severity := 4,
    VI_Active := GVL_STATE.G_Freeze_Hardware_Failed,
    VI_Timestamp := VI_System_Time_MS,
    VI_Source := 430,
    VIO_Events := GVL_STATUS.G_Diagnostics_Events,
    VIO_Count := GVL_STATUS.G_Diagnostics_Count
);

// ======================================================
// ROOT CAUSE EXPORT TO EXISTING DIAGNOSTIC FIELDS
// ======================================================
GVL_STATUS.G_Diagnostics.Subsystem_Degraded := GVL_STATUS.G_Diagnostics.Subsystem_Degraded OR L_Any_Heating_Device_Failed;
GVL_STATUS.G_Diagnostics.Freeze_Hardware_Event_Pending := GVL_STATUS.G_Diagnostics.Freeze_Hardware_Event_Pending OR L_Critical_Fault;

IF L_Any_Heating_Device_Failed THEN
    GVL_STATUS.G_Diagnostics.Freeze_Hardware_Event_Text := 'Heating device availability degraded';
END_IF;

IF L_Critical_Fault THEN
    GVL_STATUS.G_Diagnostics.Freeze_Hardware_Event_Text := 'Freeze hardware critical fault';
END_IF;

END_FUNCTION_BLOCK
// >>> BULK_SYNC_ANCHOR: FB_Heating_Diagnostics <<<

(* ---- FB_Heating_Freeze_Hardware.st ---- *)
FUNCTION_BLOCK FB_Heating_Freeze_Hardware

// Extracted candidate from PRG_Heating S5.
// Not connected yet.
// Donor logic remains in PRG_Heating until all extracted candidates are prepared.

GVL_STATE.G_Freeze_Hardware_Degraded := GVL_STATUS.G_Diagnostics.Backup_Pump_Fault OR GVL_STATUS.G_Diagnostics.Electric_Heater_Fault;
GVL_STATE.G_Freeze_Hardware_Failed := GVL_STATUS.G_Diagnostics.Backup_Pump_Fault AND GVL_STATUS.G_Diagnostics.Electric_Heater_Fault;

IF GVL_STATE.G_Freeze_Hardware_Failed THEN
    GVL_STATE.G_Backup_Circulation_Pump := FALSE;
    GVL_STATE.G_Electric_Heater_Enable := FALSE;
    GVL_STATE.G_Safety_Freeze_Risk := TRUE;
END_IF;

END_FUNCTION_BLOCK
// >>> BULK_SYNC_ANCHOR: FB_Heating_Freeze_Hardware <<<

(* ---- FB_Heating_Local_Context.st ---- *)
FUNCTION_BLOCK FB_Heating_Local_Context
VAR_INPUT
    VI_System_Time_MS : UDINT;
    VI_Safety_Emergency_Stop : BOOL;
    VI_Safety_Gas_Latched : BOOL;
    VI_DHW_Block : BOOL;
    VI_Freeze_Request : BOOL;
    VI_Preheat_Request : BOOL;
    VI_DHW_Heating_Pump_Feedback : BOOL;
    VI_Policy_Target_Adjustment : REAL;
    VI_Boiler_Modulation_Raw : ARRAY[1..GVL_CONSTANTS.C_MAX_BOILERS] OF INT;
END_VAR
VAR_OUTPUT
    VO_Boiler_Modulation_REAL : ARRAY[1..GVL_CONSTANTS.C_MAX_BOILERS] OF REAL;
    VO_Heating_Emergency_Stop : BOOL;
    VO_Heating_Gas_Safety_Stop : BOOL;
    VO_Heating_DHW_Demand : BOOL;
    VO_Target_Temperature : REAL;
    VO_Local_Mode : INT;
END_VAR
VAR
    L_Last_Mode : INT := 0; // 0=normal, 1=preheat, 2=freeze
    L_Mode_Hold_Timer : FB_System_Timer;
    L_i : INT;
END_VAR

// Local heating context builder.
// DHW blocking now comes from the command layer via VI_DHW_Block.
// Safety still gates local heating/DHW context until full safety-command migration is complete.

FOR L_i := 1 TO GVL_CONSTANTS.C_MAX_BOILERS DO
    VO_Boiler_Modulation_REAL[L_i] := TO_REAL(VI_Boiler_Modulation_Raw[L_i]);
END_FOR;

VO_Heating_Emergency_Stop := VI_Safety_Emergency_Stop;
VO_Heating_Gas_Safety_Stop := VI_Safety_Gas_Latched;
VO_Heating_DHW_Demand := VI_DHW_Heating_Pump_Feedback;

IF VO_Heating_Emergency_Stop THEN
    VO_Heating_Gas_Safety_Stop := FALSE;
    VO_Heating_DHW_Demand := FALSE;
ELSIF VO_Heating_Gas_Safety_Stop THEN
    VO_Heating_DHW_Demand := FALSE;
ELSIF VI_DHW_Block THEN
    VO_Heating_DHW_Demand := FALSE;
END_IF;

L_Mode_Hold_Timer(
    IN := TRUE,
    PT := T#30s,
    VI_System_Time_MS := VI_System_Time_MS
);

IF L_Mode_Hold_Timer.Q THEN
    IF VI_Freeze_Request THEN
        L_Last_Mode := 2;
    ELSIF VI_Preheat_Request THEN
        L_Last_Mode := 1;
    ELSE
        L_Last_Mode := 0;
    END_IF;
END_IF;

CASE L_Last_Mode OF
    2: VO_Target_Temperature := 5.0;
    1: VO_Target_Temperature := 22.0;
    ELSE VO_Target_Temperature := 20.0;
END_CASE;

VO_Target_Temperature := VO_Target_Temperature + VI_Policy_Target_Adjustment;
IF VO_Target_Temperature < 5.0 THEN
    VO_Target_Temperature := 5.0;
ELSIF VO_Target_Temperature > 26.0 THEN
    VO_Target_Temperature := 26.0;
END_IF;

VO_Local_Mode := L_Last_Mode;

END_FUNCTION_BLOCK
// >>> BULK_SYNC_ANCHOR: FB_Heating_Local_Context <<<

(* ---- FB_Heating_Manifold_Control.st ---- *)
// ==============================================================================
// Heating manifold control helper
// Internal refactoring helper for FB_Heating_System_Manager.
// Valve test override remains in FB_Heating_System_Manager for now.
// ==============================================================================
FUNCTION_BLOCK FB_Heating_Manifold_Control
VAR_INPUT
    VI_System_Time_MS : UDINT;
    VI_IsActivePLC : BOOL;
    VI_DHW_Heating_Demand : BOOL;
    VI_Freeze_Mode_Active : BOOL;
    VI_Target_Supply_Temp : REAL;
    VI_Any_Zone_Active : ARRAY[1..GVL_CONSTANTS.C_MAX_MANIFOLDS] OF BOOL;
END_VAR

VAR_IN_OUT
    VI_Manifold_Pressures : ARRAY[1..GVL_CONSTANTS.C_MAX_MANIFOLDS] OF REAL;
    VI_Manifold_Currents : ARRAY[1..GVL_CONSTANTS.C_MAX_MANIFOLDS] OF REAL;
    VI_Manifold_Temps_Supply : ARRAY[1..GVL_CONSTANTS.C_MAX_MANIFOLDS] OF REAL;
    VI_Manifold_Temps_Return : ARRAY[1..GVL_CONSTANTS.C_MAX_MANIFOLDS] OF REAL;
END_VAR

VAR_OUTPUT
    VO_Manifold_Pumps : ARRAY[1..GVL_CONSTANTS.C_MAX_MANIFOLDS] OF BOOL;
    VO_Manifold_Valves : ARRAY[1..GVL_CONSTANTS.C_MAX_MANIFOLDS] OF REAL;
    VO_Status : ARRAY[1..GVL_CONSTANTS.C_MAX_MANIFOLDS] OF ST_Manifold_Status;
END_VAR

VAR
    L_i : INT;
    L_Delta_T : REAL;
    L_PID_Valves : ARRAY[1..GVL_CONSTANTS.C_MAX_MANIFOLDS] OF FB_PID_Controller;
    L_PID_Timer : ARRAY[1..GVL_CONSTANTS.C_MAX_MANIFOLDS] OF FB_System_Timer;
    L_Pump_Run_Timer : ARRAY[1..GVL_CONSTANTS.C_MAX_MANIFOLDS] OF FB_System_Timer;
    L_Pump_Pause_Timer : ARRAY[1..GVL_CONSTANTS.C_MAX_MANIFOLDS] OF FB_System_Timer;
    L_Pump_In_Pause : ARRAY[1..GVL_CONSTANTS.C_MAX_MANIFOLDS] OF BOOL;
    L_Pump_Diag : ARRAY[1..GVL_CONSTANTS.C_MAX_MANIFOLDS] OF FB_Device_Predictive_Diag;
END_VAR

FOR L_i := 1 TO GVL_CONSTANTS.C_MAX_MANIFOLDS DO
    L_PID_Timer[L_i](IN := TRUE, PT := T#1s, VI_System_Time_MS := VI_System_Time_MS);
    IF L_PID_Timer[L_i].Q THEN
        L_PID_Timer[L_i](IN := FALSE, PT := T#1s, VI_System_Time_MS := VI_System_Time_MS);
        L_PID_Timer[L_i](IN := TRUE, PT := T#1s, VI_System_Time_MS := VI_System_Time_MS);

        L_PID_Valves[L_i](
            VI_SetPoint := VI_Target_Supply_Temp,
            VI_ProcessValue := VI_Manifold_Temps_Supply[L_i],
            VI_Kp := 2.0,
            VI_Tn := 120.0,
            VI_Tv := 0.0,
            VI_Y_Min := 0.0,
            VI_Y_Max := 100.0,
            VI_Cycle_Time_S := 1.0,
            VO_Output => VO_Manifold_Valves[L_i]
        );
    END_IF;

    L_Pump_Run_Timer[L_i](
        IN := VO_Manifold_Pumps[L_i] AND NOT L_Pump_In_Pause[L_i],
        PT := T#72h,
        VI_System_Time_MS := VI_System_Time_MS
    );
    IF L_Pump_Run_Timer[L_i].Q THEN
        L_Pump_In_Pause[L_i] := TRUE;
    END_IF;

    L_Pump_Pause_Timer[L_i](
        IN := L_Pump_In_Pause[L_i],
        PT := T#1h,
        VI_System_Time_MS := VI_System_Time_MS
    );
    IF L_Pump_Pause_Timer[L_i].Q THEN
        L_Pump_In_Pause[L_i] := FALSE;
    END_IF;

    IF VI_DHW_Heating_Demand THEN
        VO_Manifold_Pumps[L_i] := FALSE;
        VO_Manifold_Valves[L_i] := 0.0;
    ELSE
        VO_Manifold_Pumps[L_i] := VI_IsActivePLC AND VI_Any_Zone_Active[L_i] AND NOT L_Pump_In_Pause[L_i];
    END_IF;

    IF VI_Freeze_Mode_Active THEN
        VO_Manifold_Pumps[L_i] := TRUE;
        IF VO_Manifold_Valves[L_i] < 35.0 THEN
            VO_Manifold_Valves[L_i] := 35.0;
        END_IF;
    END_IF;

    VO_Status[L_i].Pump_On := VO_Manifold_Pumps[L_i];
    VO_Status[L_i].Pump_Current := VI_Manifold_Currents[L_i];
    VO_Status[L_i].Pressure := VI_Manifold_Pressures[L_i];
    VO_Status[L_i].Temp_Supply := VI_Manifold_Temps_Supply[L_i];
    VO_Status[L_i].Temp_Return := VI_Manifold_Temps_Return[L_i];
    VO_Status[L_i].Valve_Pos := VO_Manifold_Valves[L_i];

    L_Pump_Diag[L_i](
        VI_Current_Value := VI_Manifold_Currents[L_i],
        VI_Nominal_Value := 0.55,
        VI_Is_Running := VO_Manifold_Pumps[L_i],
        VI_Reset_Stats := FALSE,
        VI_System_Time_MS := VI_System_Time_MS,
        VIO_Health_Data := VO_Status[L_i].Health
    );

    IF VO_Manifold_Pumps[L_i] THEN
        L_Delta_T := VI_Manifold_Temps_Supply[L_i] - VI_Manifold_Temps_Return[L_i];

        VO_Status[L_i].Error := FALSE;
        VO_Status[L_i].Error_ID := 0;

        IF VI_Manifold_Currents[L_i] <= 0.01 THEN
            VO_Status[L_i].Error := TRUE;
            VO_Status[L_i].Error_ID := TO_WORD(GVL_CONFIG.ERR_PUMP_NO_CURRENT);
        ELSIF VI_Manifold_Currents[L_i] < 0.3 THEN
            VO_Status[L_i].Error := TRUE;
            VO_Status[L_i].Error_ID := TO_WORD(GVL_CONFIG.ERR_PUMP_UNDERCURRENT);
        ELSIF VI_Manifold_Currents[L_i] > 1.5 THEN
            VO_Status[L_i].Error := TRUE;
            VO_Status[L_i].Error_ID := TO_WORD(GVL_CONFIG.ERR_PUMP_OVERCURRENT);
        END_IF;

        IF (NOT VO_Status[L_i].Error) AND ((VI_Manifold_Pressures[L_i] < 1.5) OR (VI_Manifold_Pressures[L_i] > 2.5)) THEN
            VO_Status[L_i].Error := TRUE;
            VO_Status[L_i].Error_ID := TO_WORD(GVL_CONFIG.ERR_PRESSURE_OUT_OF_RANGE);
        END_IF;

        IF NOT VO_Status[L_i].Error THEN
            IF L_Delta_T < 5.0 THEN
                VO_Status[L_i].Error := TRUE;
                VO_Status[L_i].Error_ID := TO_WORD(GVL_CONFIG.ERR_DELTA_T_LOW);
            ELSIF L_Delta_T > 10.0 THEN
                VO_Status[L_i].Error := TRUE;
                VO_Status[L_i].Error_ID := TO_WORD(GVL_CONFIG.ERR_DELTA_T_HIGH);
            END_IF;
        END_IF;
    END_IF;
END_FOR;

// >>> BULK_SYNC_ANCHOR: FB_Heating_Manifold_Control <<<

(* ---- FB_Heating_Orchestration.st ---- *)
FUNCTION_BLOCK FB_Heating_Orchestration
VAR_INPUT
    VI_System_Time_MS : UDINT;
    VI_Current_TOD : TOD;
    VI_Current_Day_Of_Week : UINT;
    VI_IsActivePLC : BOOL;
    VI_Outdoor_Temp : REAL;
    VI_Floor_Temps : ARRAY[1..GVL_CONSTANTS.C_MAX_HEATING_CIRCUITS] OF REAL;
    VI_Room_Temps : ARRAY[1..GVL_CONSTANTS.C_MAX_ZONES] OF REAL;
    VI_Config : ST_Heating_Config;
    VI_Zone_Configs : ARRAY[1..GVL_CONSTANTS.C_MAX_HEATING_CIRCUITS] OF ST_FloorHeating_Circuit_Config;
    VI_Tariff : ST_Tariff_Config;
    VI_Time_Of_Day_MS : UDINT;
    VI_Manifold_Pressures : ARRAY[1..GVL_CONSTANTS.C_MAX_MANIFOLDS] OF REAL;
    VI_Manifold_Currents : ARRAY[1..GVL_CONSTANTS.C_MAX_MANIFOLDS] OF REAL;
    VI_Manifold_Temps_Supply : ARRAY[1..GVL_CONSTANTS.C_MAX_MANIFOLDS] OF REAL;
    VI_Manifold_Temps_Return : ARRAY[1..GVL_CONSTANTS.C_MAX_MANIFOLDS] OF REAL;
    VI_Boiler_Flame_Status : ARRAY[1..GVL_CONSTANTS.C_MAX_BOILERS] OF BOOL;
    VI_Boiler_Error_Status : ARRAY[1..GVL_CONSTANTS.C_MAX_BOILERS] OF BOOL;
    VI_Boiler_OT_Online : ARRAY[1..GVL_CONSTANTS.C_MAX_BOILERS] OF BOOL;
    VI_Boiler_Modulation : ARRAY[1..GVL_CONSTANTS.C_MAX_BOILERS] OF REAL;
    VI_Rule_Actions : ARRAY[1..GVL_CONSTANTS.C_MAX_RULES] OF ST_Rule_Action;
    VI_IO_Modules_Online : ARRAY[1..GVL_CONSTANTS.C_MAX_MODULES] OF BOOL;
    VI_DHW_Heating_Demand : BOOL;
    VI_DHW_Target_Temp : REAL;
    VI_DHW_Temp : REAL;
    VI_DHW_Pressure : REAL;
    VI_DHW_Config : ST_DHW_Config;
    VI_Reset_Errors : BOOL;
    VI_System_Mode : E_System_Operating_Mode;
    VI_Emergency_Stop : BOOL;
    VI_Gas_Safety_Stop : BOOL;
    VI_Manifold_End_Switches : ARRAY[1..GVL_CONSTANTS.C_MAX_MANIFOLDS] OF BOOL;
    VI_Valve_Test_Config : ARRAY[1..GVL_CONSTANTS.C_MAX_MANIFOLDS] OF ST_Valve_Test_Config;
    VI_Block_Heating : BOOL;
    VI_Manifold_Enabled : ARRAY[1..GVL_CONSTANTS.C_MAX_MANIFOLDS] OF BOOL;
END_VAR
VAR_IN_OUT
    VIO_Manifold_Valves : ARRAY[1..GVL_CONSTANTS.C_MAX_MANIFOLDS] OF REAL;
    VIO_Manifold_Pumps : ARRAY[1..GVL_CONSTANTS.C_MAX_MANIFOLDS] OF BOOL;
    VIO_Zone_Valves : ARRAY[1..GVL_CONSTANTS.C_MAX_HEATING_CIRCUITS] OF BOOL;
    VIO_Boiler_OT_Enable : ARRAY[1..GVL_CONSTANTS.C_MAX_BOILERS] OF BOOL;
    VIO_Boiler_OT_Setpoint : ARRAY[1..GVL_CONSTANTS.C_MAX_BOILERS] OF REAL;
    VIO_Backup_Circulation_Pump : BOOL;
    VIO_Electric_Heater_Enable : BOOL;
    VIO_Freeze_Risk_Status : BOOL;
    VIO_Manifold_Status : ARRAY[1..GVL_CONSTANTS.C_MAX_MANIFOLDS] OF ST_Manifold_Status;
    VIO_Boiler_Status : ARRAY[1..GVL_CONSTANTS.C_MAX_BOILERS] OF ST_Boiler_Status;
    VIO_DHW_Heating_Pump : BOOL;
    VIO_DHW_Circ_Pump : BOOL;
    VIO_DHW_Status : ST_DHW_Status;
END_VAR
VAR
    fbHeatingManager : FB_Heating_System_Manager;
    fbDHWManager : FB_DHW_Manager;
    L_i : INT;
    L_j : INT;
END_VAR

// Extracted candidate from PRG_Heating S2.
// Not connected yet.
// Donor logic remains in PRG_Heating until all extracted candidates are prepared.

fbHeatingManager(
    VI_System_Time_MS := VI_System_Time_MS,
    VI_IsActivePLC := VI_IsActivePLC,
    VI_Outdoor_Temp := VI_Outdoor_Temp,
    VI_Floor_Temps := VI_Floor_Temps,
    VI_Room_Temps := VI_Room_Temps,
    VI_Config := VI_Config,
    VI_Zone_Configs := VI_Zone_Configs,
    VI_Tariff := VI_Tariff,
    VI_Current_Hour := TO_UINT(VI_Time_Of_Day_MS / GVL_CONSTANTS.C_MS_IN_HOUR),
    VI_Manifold_Pressures := VI_Manifold_Pressures,
    VI_Manifold_Currents := VI_Manifold_Currents,
    VI_Manifold_Temps_Supply := VI_Manifold_Temps_Supply,
    VI_Manifold_Temps_Return := VI_Manifold_Temps_Return,
    VI_Boiler_Flame_Status := VI_Boiler_Flame_Status,
    VI_Boiler_Error_Status := VI_Boiler_Error_Status,
    VI_Boiler_OT_Online := VI_Boiler_OT_Online,
    VI_Boiler_Modulation := VI_Boiler_Modulation,
    VI_Rule_Actions := VI_Rule_Actions,
    VI_IO_Modules_Online := VI_IO_Modules_Online,
    VI_DHW_Heating_Demand := VI_DHW_Heating_Demand,
    VI_DHW_Target_Temp := VI_DHW_Target_Temp,
    VI_System_Mode := VI_System_Mode,
    VI_Emergency_Stop := VI_Emergency_Stop,
    VI_Gas_Safety_Stop := VI_Gas_Safety_Stop,
    VI_Manifold_End_Switches := VI_Manifold_End_Switches,
    VI_Valve_Test_Config := VI_Valve_Test_Config,
    VO_Manifold_Valves => VIO_Manifold_Valves,
    VO_Manifold_Pumps => VIO_Manifold_Pumps,
    VO_Zone_Valves => VIO_Zone_Valves,
    VO_Boiler_OT_Enable => VIO_Boiler_OT_Enable,
    VO_Boiler_OT_Setpoint => VIO_Boiler_OT_Setpoint,
    VO_Backup_Circulation_Pump => VIO_Backup_Circulation_Pump,
    VO_Electric_Heater_Enable => VIO_Electric_Heater_Enable,
    VO_Freeze_Risk_Status => VIO_Freeze_Risk_Status,
    VO_Status => VIO_Manifold_Status,
    VO_Boiler_Status => VIO_Boiler_Status
);

FOR L_i := 1 TO GVL_CONSTANTS.C_MAX_MANIFOLDS DO
    IF VI_Block_Heating OR (NOT VI_Manifold_Enabled[L_i]) THEN
        VIO_Manifold_Pumps[L_i] := FALSE;
        VIO_Manifold_Valves[L_i] := 0.0;

        FOR L_j := 1 TO GVL_CONSTANTS.C_MAX_HEATING_CIRCUITS DO
            IF VI_Zone_Configs[L_j].manifold_id = L_i THEN
                VIO_Zone_Valves[L_j] := FALSE;
            END_IF;
        END_FOR;
    END_IF;
END_FOR;

fbDHWManager(
    VI_System_Time_MS := VI_System_Time_MS,
    VI_Current_TOD := VI_Current_TOD,
    VI_IsActivePLC := VI_IsActivePLC,
    VI_Temp := VI_DHW_Temp,
    VI_Pressure := VI_DHW_Pressure,
    VI_Config := VI_DHW_Config,
    VI_Current_Day_Of_Week := VI_Current_Day_Of_Week,
    VI_IO_Modules_Online := VI_IO_Modules_Online,
    VI_Reset_Errors := VI_Reset_Errors,
    VI_Emergency_Stop := VI_Emergency_Stop,
    VI_System_Mode := VI_System_Mode,
    VO_Heating_Pump => VIO_DHW_Heating_Pump,
    VO_Circ_Pump => VIO_DHW_Circ_Pump,
    VO_Status => VIO_DHW_Status
);

END_FUNCTION_BLOCK
// >>> BULK_SYNC_ANCHOR: FB_Heating_Orchestration <<<

(* ---- FB_Heating_Output_Projection.st ---- *)
FUNCTION_BLOCK FB_Heating_Output_Projection
VAR_INPUT
    VI_Zone_Valves : ARRAY[1..8] OF BOOL;
    VI_Manifold_Pumps : ARRAY[1..GVL_CONSTANTS.C_MAX_MANIFOLDS] OF BOOL;
    VI_Manifold_Valves : ARRAY[1..GVL_CONSTANTS.C_MAX_MANIFOLDS] OF REAL;
    VI_DHW_Heating_Pump : BOOL;
    VI_DHW_Circ_Pump : BOOL;
    VI_Backup_Circulation_Pump : BOOL;
    VI_Electric_Heater_Enable : BOOL;
END_VAR
VAR
    L_i : INT;
END_VAR

// Converts STATE-level outputs into IO-ready projection (no commands applied here).

FOR L_i := 1 TO 8 DO
    GVL_HEATING_OUTPUT.DO_Zone_Valves[L_i] := VI_Zone_Valves[L_i];
END_FOR;

FOR L_i := 1 TO GVL_CONSTANTS.C_MAX_MANIFOLDS DO
    GVL_HEATING_OUTPUT.DO_Manifold_Pumps[L_i] := VI_Manifold_Pumps[L_i];
    GVL_HEATING_OUTPUT.AO_Manifold_Valves[L_i] := REAL_TO_UINT(VI_Manifold_Valves[L_i] * 1000.0);
END_FOR;

GVL_HEATING_OUTPUT.DO_DHW_Heating_Pump := VI_DHW_Heating_Pump;
GVL_HEATING_OUTPUT.DO_DHW_Circ_Pump := VI_DHW_Circ_Pump;
GVL_HEATING_OUTPUT.DO_Backup_Circulation_Pump := VI_Backup_Circulation_Pump;
GVL_HEATING_OUTPUT.DO_Electric_Heater_Enable := VI_Electric_Heater_Enable;

END_FUNCTION_BLOCK
// >>> BULK_SYNC_ANCHOR: FB_Heating_Output_Projection <<<

(* ---- FB_Heating_Override_Layer.st ---- *)
FUNCTION_BLOCK FB_Heating_Override_Layer
VAR_INPUT
    VI_Block_Heating : BOOL;
    VI_Manifold_Enabled : ARRAY[1..GVL_CONSTANTS.C_MAX_MANIFOLDS] OF BOOL;
    VI_Zone_Configs : ARRAY[1..GVL_CONSTANTS.C_MAX_HEATING_CIRCUITS] OF ST_FloorHeating_Circuit_Config;
END_VAR
VAR_IN_OUT
    VIO_Manifold_Valves : ARRAY[1..GVL_CONSTANTS.C_MAX_MANIFOLDS] OF REAL;
    VIO_Manifold_Pumps : ARRAY[1..GVL_CONSTANTS.C_MAX_MANIFOLDS] OF BOOL;
    VIO_Zone_Valves : ARRAY[1..GVL_CONSTANTS.C_MAX_HEATING_CIRCUITS] OF BOOL;
    VIO_Boiler_OT_Enable : ARRAY[1..GVL_CONSTANTS.C_MAX_BOILERS] OF BOOL;
    VIO_Boiler_OT_Setpoint : ARRAY[1..GVL_CONSTANTS.C_MAX_BOILERS] OF REAL;
    VIO_Backup_Circulation_Pump : BOOL;
    VIO_Electric_Heater_Enable : BOOL;
    VIO_DHW_Heating_Pump : BOOL;
    VIO_DHW_Circ_Pump : BOOL;
END_VAR
VAR
    L_i : INT;
    L_j : INT;
END_VAR

FOR L_i := 1 TO GVL_CONSTANTS.C_MAX_MANIFOLDS DO
    IF VI_Block_Heating OR (NOT VI_Manifold_Enabled[L_i]) THEN
        VIO_Manifold_Pumps[L_i] := FALSE;
        VIO_Manifold_Valves[L_i] := 0.0;

        FOR L_j := 1 TO GVL_CONSTANTS.C_MAX_HEATING_CIRCUITS DO
            IF VI_Zone_Configs[L_j].manifold_id = L_i THEN
                VIO_Zone_Valves[L_j] := FALSE;
            END_IF;
        END_FOR;
    END_IF;
END_FOR;

IF VI_Block_Heating THEN
    FOR L_i := 1 TO GVL_CONSTANTS.C_MAX_HEATING_CIRCUITS DO
        VIO_Zone_Valves[L_i] := FALSE;
    END_FOR;

    FOR L_i := 1 TO GVL_CONSTANTS.C_MAX_MANIFOLDS DO
        VIO_Manifold_Pumps[L_i] := FALSE;
        VIO_Manifold_Valves[L_i] := 0.0;
    END_FOR;

    FOR L_i := 1 TO GVL_CONSTANTS.C_MAX_BOILERS DO
        VIO_Boiler_OT_Enable[L_i] := FALSE;
        VIO_Boiler_OT_Setpoint[L_i] := 0.0;
    END_FOR;

    VIO_Backup_Circulation_Pump := FALSE;
    VIO_Electric_Heater_Enable := FALSE;
    VIO_DHW_Heating_Pump := FALSE;
    VIO_DHW_Circ_Pump := FALSE;
END_IF;

END_FUNCTION_BLOCK
// >>> BULK_SYNC_ANCHOR: FB_Heating_Override_Layer <<<

(* ---- FB_Heating_Policy_Manager.st ---- *)
FUNCTION_BLOCK FB_Heating_Policy_Manager
VAR_INPUT
    VI_System_Mode : E_System_Operating_Mode;
    VI_RootCause : E_Heating_RootCause;
    VI_Emergency_Stop : BOOL;
    VI_Gas_Safety : BOOL;
END_VAR

VAR_OUTPUT
    VO_Policy_Mode : E_Heating_Policy_Mode;
    VO_Block_Heating : BOOL;
    VO_Target_Adjustment : REAL;
    VO_Priority_Multiplier : REAL;
END_VAR

// defaults
VO_Target_Adjustment := 0.0;
VO_Priority_Multiplier := 1.0;

// Safety has absolute priority
IF VI_Emergency_Stop OR VI_Gas_Safety THEN
    VO_Policy_Mode := E_Heating_Policy_Mode.HPM_SAFETY_BLOCK;
    VO_Block_Heating := TRUE;
    RETURN;
END_IF;

// Root cause driven policy
CASE VI_RootCause OF

    E_Heating_RootCause.RC_IO_OFFLINE:
        VO_Policy_Mode := E_Heating_Policy_Mode.HPM_DEGRADED;
        VO_Block_Heating := TRUE;
        RETURN;

    E_Heating_RootCause.RC_PUMP_FAILURE:
        VO_Policy_Mode := E_Heating_Policy_Mode.HPM_FAULT_ISOLATION;
        VO_Priority_Multiplier := 0.5; // reduce load
        RETURN;

    E_Heating_RootCause.RC_VALVES_CLOSED:
        VO_Policy_Mode := E_Heating_Policy_Mode.HPM_FAULT_ISOLATION;
        VO_Target_Adjustment := -2.0;
        RETURN;

    E_Heating_RootCause.RC_NO_HEAT_TRANSFER:
        VO_Policy_Mode := E_Heating_Policy_Mode.HPM_DEGRADED;
        VO_Target_Adjustment := +3.0;
        RETURN;

    E_Heating_RootCause.RC_NO_FLAME,
    E_Heating_RootCause.RC_BOILER_ERROR:
        VO_Policy_Mode := E_Heating_Policy_Mode.HPM_DEGRADED;
        VO_Priority_Multiplier := 0.7;
        RETURN;

END_CASE;

// System mode fallback
IF VI_System_Mode = E_System_Operating_Mode.MODE_DEGRADED THEN
    VO_Policy_Mode := E_Heating_Policy_Mode.HPM_DEGRADED;
ELSE
    VO_Policy_Mode := E_Heating_Policy_Mode.HPM_NORMAL;
END_IF;

VO_Block_Heating := FALSE;

END_FUNCTION_BLOCK

(* ---- FB_Heating_Policy_Observer.st ---- *)
FUNCTION_BLOCK FB_Heating_Policy_Observer

VAR_INPUT
    VI_Zone_Occupied : ARRAY[1..GVL_CONSTANTS.C_MAX_ZONES] OF BOOL;
    VI_Zone_Last_Motion_TS : ARRAY[1..GVL_CONSTANTS.C_MAX_ZONES] OF UDINT;
    VI_System_Time_MS : UDINT;
    VI_Zone_Permanent_Use : ARRAY[1..GVL_CONSTANTS.C_MAX_ZONES] OF BOOL;
    VI_Zone_Guest_Preheat : ARRAY[1..GVL_CONSTANTS.C_MAX_ZONES] OF BOOL;
    VI_Behavior_Mode : E_Behavior_Mode;
END_VAR

VAR_OUTPUT
    VO_Zone_Empty_Duration_MS : ARRAY[1..GVL_CONSTANTS.C_MAX_ZONES] OF UDINT;
    VO_Zone_Policy_Class : ARRAY[1..GVL_CONSTANTS.C_MAX_ZONES] OF INT;
    VO_Zone_Target_Adjustment : ARRAY[1..GVL_CONSTANTS.C_MAX_ZONES] OF REAL;
    VO_Zone_Priority_Bias : ARRAY[1..GVL_CONSTANTS.C_MAX_ZONES] OF REAL;
END_VAR

VAR
    L_i : INT;
    L_Long_Threshold : UDINT := 86400000; // 24h
    L_Away_Mode : BOOL;
END_VAR

L_Away_Mode := (VI_Behavior_Mode = BEHAVIOR_AWAY);

FOR L_i := 1 TO GVL_CONSTANTS.C_MAX_ZONES DO

    // compute empty duration
    IF VI_Zone_Occupied[L_i] THEN
        VO_Zone_Empty_Duration_MS[L_i] := 0;
    ELSE
        VO_Zone_Empty_Duration_MS[L_i] := VI_System_Time_MS - VI_Zone_Last_Motion_TS[L_i];
    END_IF;

    // policy classification
    // Guest/preheat has priority even in AWAY mode.
    IF VI_Zone_Guest_Preheat[L_i] THEN
        VO_Zone_Policy_Class[L_i] := 3; // guest

    ELSIF VI_Zone_Occupied[L_i] THEN
        VO_Zone_Policy_Class[L_i] := 0; // comfort

    ELSIF VI_Zone_Permanent_Use[L_i] AND (NOT L_Away_Mode) THEN
        VO_Zone_Policy_Class[L_i] := 4; // permanent mild eco

    ELSIF VO_Zone_Empty_Duration_MS[L_i] >= L_Long_Threshold THEN
        VO_Zone_Policy_Class[L_i] := 2; // deep eco

    ELSE
        VO_Zone_Policy_Class[L_i] := 1; // mild eco
    END_IF;

    // observe-only target adjustment (no effect yet)
    CASE VO_Zone_Policy_Class[L_i] OF
        0: // comfort
            VO_Zone_Target_Adjustment[L_i] := 0.0;
            VO_Zone_Priority_Bias[L_i] := 1.0;

        1: // mild eco
            VO_Zone_Target_Adjustment[L_i] := -1.0;
            VO_Zone_Priority_Bias[L_i] := 0.8;

        2: // deep eco
            VO_Zone_Target_Adjustment[L_i] := -3.0;
            VO_Zone_Priority_Bias[L_i] := 0.5;

        3: // guest preheat
            VO_Zone_Target_Adjustment[L_i] := 0.0;
            VO_Zone_Priority_Bias[L_i] := 1.5;

        4: // permanent-use mild eco
            VO_Zone_Target_Adjustment[L_i] := -0.5;
            VO_Zone_Priority_Bias[L_i] := 0.9;

    END_CASE;

END_FOR;

(* ---- FB_Heating_Policy_Priority_Bridge.st ---- *)
// ==============================================================================
// Heating policy priority bridge
//
// Bounded mapper from advisory zone policy to manifold allocation priority.
//
// IMPORTANT:
// - does NOT own demand;
// - does NOT create demand;
// - does NOT control pumps/valves;
// - does NOT write outputs;
// - does NOT bypass safety or service gates.
//
// Responsibility:
// - map circuit->zone policy bias into manifold effective priority;
// - keep the result bounded and deterministic;
// - provide a safe input for FB_Heating_Allocation_Filter.
// ==============================================================================
FUNCTION_BLOCK FB_Heating_Policy_Priority_Bridge
VAR_INPUT
    VI_Enable : BOOL;

    VI_Zone_Valves : ARRAY[1..GVL_CONSTANTS.C_MAX_HEATING_CIRCUITS] OF BOOL;
    VI_Zone_Configs : ARRAY[1..GVL_CONSTANTS.C_MAX_HEATING_CIRCUITS] OF ST_FloorHeating_Circuit_Config;

    VI_Manifold_Base_Priority : ARRAY[1..GVL_CONSTANTS.C_MAX_MANIFOLDS] OF INT;
    VI_Zone_Priority_Bias : ARRAY[1..GVL_CONSTANTS.C_MAX_ZONES] OF REAL;
    VI_Policy_Priority_Multiplier : REAL;
END_VAR
VAR_OUTPUT
    VO_Manifold_Effective_Priority : ARRAY[1..GVL_CONSTANTS.C_MAX_MANIFOLDS] OF INT;
    VO_Manifold_Priority_Bias_Applied : ARRAY[1..GVL_CONSTANTS.C_MAX_MANIFOLDS] OF REAL;
    VO_Bridge_Active : BOOL;
END_VAR
VAR
    L_i : INT;
    L_Manifold_ID : INT;
    L_Zone_ID : INT;
    L_Multiplier : REAL;
    L_Bias : REAL;
    L_Score : REAL;
    L_MaxScore : ARRAY[1..GVL_CONSTANTS.C_MAX_MANIFOLDS] OF REAL;
    L_HasActiveCircuit : ARRAY[1..GVL_CONSTANTS.C_MAX_MANIFOLDS] OF BOOL;
END_VAR

// Default passthrough state.
VO_Bridge_Active := FALSE;

FOR L_i := 1 TO GVL_CONSTANTS.C_MAX_MANIFOLDS DO
    VO_Manifold_Effective_Priority[L_i] := VI_Manifold_Base_Priority[L_i];
    VO_Manifold_Priority_Bias_Applied[L_i] := REAL#1.0;
    L_MaxScore[L_i] := REAL#0.0;
    L_HasActiveCircuit[L_i] := FALSE;
END_FOR;

IF NOT VI_Enable THEN
    RETURN;
END_IF;

L_Multiplier := VI_Policy_Priority_Multiplier;
IF L_Multiplier < REAL#0.3 THEN
    L_Multiplier := REAL#0.3;
ELSIF L_Multiplier > REAL#1.0 THEN
    L_Multiplier := REAL#1.0;
END_IF;

IF ABS(L_Multiplier - REAL#1.0) > REAL#0.001 THEN
    VO_Bridge_Active := TRUE;
END_IF;

FOR L_i := 1 TO GVL_CONSTANTS.C_MAX_HEATING_CIRCUITS DO
    IF VI_Zone_Valves[L_i] THEN
        L_Manifold_ID := TO_INT(VI_Zone_Configs[L_i].manifold_id);
        L_Zone_ID := TO_INT(VI_Zone_Configs[L_i].zone);

        IF (L_Manifold_ID >= 1)
           AND (L_Manifold_ID <= GVL_CONSTANTS.C_MAX_MANIFOLDS)
           AND (L_Zone_ID >= 1)
           AND (L_Zone_ID <= GVL_CONSTANTS.C_MAX_ZONES) THEN

            L_Bias := VI_Zone_Priority_Bias[L_Zone_ID];
            IF L_Bias < REAL#0.3 THEN
                L_Bias := REAL#0.3;
            ELSIF L_Bias > REAL#1.5 THEN
                L_Bias := REAL#1.5;
            END_IF;

            IF ABS(L_Bias - REAL#1.0) > REAL#0.001 THEN
                VO_Bridge_Active := TRUE;
            END_IF;

            IF L_Bias > VO_Manifold_Priority_Bias_Applied[L_Manifold_ID] THEN
                VO_Manifold_Priority_Bias_Applied[L_Manifold_ID] := L_Bias;
            END_IF;

            L_Score := TO_REAL(VI_Manifold_Base_Priority[L_Manifold_ID]) * L_Multiplier * L_Bias;

            IF L_Score > L_MaxScore[L_Manifold_ID] THEN
                L_MaxScore[L_Manifold_ID] := L_Score;
            END_IF;

            L_HasActiveCircuit[L_Manifold_ID] := TRUE;
        END_IF;
    END_IF;
END_FOR;

FOR L_i := 1 TO GVL_CONSTANTS.C_MAX_MANIFOLDS DO
    IF L_HasActiveCircuit[L_i] THEN
        IF L_MaxScore[L_i] >= REAL#3.5 THEN
            VO_Manifold_Effective_Priority[L_i] := 4;
        ELSIF L_MaxScore[L_i] >= REAL#2.5 THEN
            VO_Manifold_Effective_Priority[L_i] := 3;
        ELSIF L_MaxScore[L_i] >= REAL#1.5 THEN
            VO_Manifold_Effective_Priority[L_i] := 2;
        ELSIF L_MaxScore[L_i] >= REAL#0.5 THEN
            VO_Manifold_Effective_Priority[L_i] := 1;
        ELSE
            VO_Manifold_Effective_Priority[L_i] := 0;
        END_IF;
    ELSE
        VO_Manifold_Effective_Priority[L_i] := VI_Manifold_Base_Priority[L_i];
        VO_Manifold_Priority_Bias_Applied[L_i] := REAL#1.0;
    END_IF;
END_FOR;

END_FUNCTION_BLOCK
// >>> BULK_SYNC_ANCHOR: FB_Heating_Policy_Priority_Bridge <<<

(* ---- FB_Heating_RootCause_Diagnostics.st ---- *)
// ==============================================================================
// Heating root-cause diagnostics observer
// Pure diagnostics/explainability layer.
// Does NOT own control/runtime decisions.
// ==============================================================================
FUNCTION_BLOCK FB_Heating_RootCause_Diagnostics
VAR_INPUT
    VI_Enable : BOOL;
END_VAR
VAR
    L_RootCause : E_Heating_RootCause;
    L_Confidence : REAL;
    L_Confidence_Text : STRING(128);
    L_Confidence_Code : INT;
END_VAR

// ======================================================
// DEFAULTS
// ======================================================
L_RootCause := E_Heating_RootCause.RC_NONE;
L_Confidence := 1.0;
L_Confidence_Text := 'Heating operating normally';
L_Confidence_Code := 0;

IF NOT VI_Enable THEN
    GVL_STATE.G_Heating_RootCause := E_Heating_RootCause.RC_NONE;
    GVL_STATE.G_Heating_RootConfidence := 0.0;
    GVL_STATE.G_Heating_Confidence := 0.0;
    GVL_STATE.G_Heating_Error_Score := 1.0;
    GVL_STATE.G_Heating_Confidence_Reason_Code := -1;
    GVL_STATE.G_Heating_Confidence_Reason_Text := 'Heating diagnostics disabled';
    RETURN;
END_IF;

// ======================================================
// ROOT CAUSE PRIORITY TREE
// ======================================================
IF GVL_STATE.G_Safety_Emergency_Stop THEN

    L_RootCause := E_Heating_RootCause.RC_EMERGENCY_STOP;
    L_Confidence := 0.01;
    L_Confidence_Text := 'Heating blocked by emergency stop';
    L_Confidence_Code := 10;

ELSIF GVL_STATE.G_Safety_Gas_Latched THEN

    L_RootCause := E_Heating_RootCause.RC_GAS_SAFETY;
    L_Confidence := 0.01;
    L_Confidence_Text := 'Heating blocked by gas safety latch';
    L_Confidence_Code := 20;

ELSIF GVL_STATE.G_Heating_IO_Fault THEN

    L_RootCause := E_Heating_RootCause.RC_IO_OFFLINE;
    L_Confidence := 0.10;
    L_Confidence_Text := 'Heating IO fault active';
    L_Confidence_Code := 30;

ELSIF NOT GVL_STATE.G_Heating_Cascade_Available THEN

    L_RootCause := E_Heating_RootCause.RC_BOILER_OFFLINE;
    L_Confidence := 0.05;
    L_Confidence_Text := 'Heating cascade unavailable';
    L_Confidence_Code := 100;

ELSIF GVL_STATE.G_Heating_Cascade_Transport_Degraded THEN

    L_RootCause := E_Heating_RootCause.RC_IO_OFFLINE;
    L_Confidence := 0.25;
    L_Confidence_Text := 'OpenTherm transport degraded';
    L_Confidence_Code := 200;

ELSIF GVL_STATE.G_Heating_Cascade_Ignition_Timeout THEN

    L_RootCause := E_Heating_RootCause.RC_NO_FLAME;
    L_Confidence := 0.20;
    L_Confidence_Text := 'Boiler ignition timeout detected';
    L_Confidence_Code := 300;

ELSIF GVL_STATE.G_Heating_Cascade_No_Flame THEN

    L_RootCause := E_Heating_RootCause.RC_NO_FLAME;
    L_Confidence := 0.35;
    L_Confidence_Text := 'Cascade active but flame missing';
    L_Confidence_Code := 400;

ELSIF GVL_STATE.G_Heating_Sensor_Fault THEN

    L_RootCause := E_Heating_RootCause.RC_SENSOR_ERROR;
    L_Confidence := 0.40;
    L_Confidence_Text := 'Heating sensor fault active';
    L_Confidence_Code := 450;

ELSIF GVL_STATE.G_Heating_Cascade_Partial_Capacity THEN

    L_RootCause := E_Heating_RootCause.RC_LOW_SUPPLY_TEMP;
    L_Confidence := 0.60;
    L_Confidence_Text := 'Partial cascade capacity available';
    L_Confidence_Code := 500;

ELSIF GVL_STATE.G_Heating_Subsystem_Degraded THEN

    L_RootCause := E_Heating_RootCause.RC_UNKNOWN;
    L_Confidence := 0.70;
    L_Confidence_Text := 'Heating subsystem degraded';
    L_Confidence_Code := 600;

ELSE

    L_RootCause := E_Heating_RootCause.RC_NONE;
    L_Confidence := 1.0;
    L_Confidence_Text := 'Heating operating normally';
    L_Confidence_Code := 0;

END_IF;

// ======================================================
// PUBLISH DIAGNOSTICS STATE
// ======================================================
GVL_STATE.G_Heating_RootCause := L_RootCause;
GVL_STATE.G_Heating_RootConfidence := L_Confidence;
GVL_STATE.G_Heating_Confidence := L_Confidence;
GVL_STATE.G_Heating_Error_Score := 1.0 - L_Confidence;
GVL_STATE.G_Heating_Confidence_Reason_Code := L_Confidence_Code;
GVL_STATE.G_Heating_Confidence_Reason_Text := L_Confidence_Text;

END_FUNCTION_BLOCK
// >>> BULK_SYNC_ANCHOR: FB_Heating_RootCause_Diagnostics <<<

(* ---- FB_Heating_Runtime_Adaptive_Drift_Detector.st ---- *)
// ==============================================================================
// Heating runtime adaptive drift detector
// Read-only adaptive supervision drift analysis layer.
// ==============================================================================
FUNCTION_BLOCK FB_Heating_Runtime_Adaptive_Drift_Detector
VAR_INPUT
    VI_Enable : BOOL;
    VI_Runtime_Risk : UINT;
    VI_Runtime_Stability : UINT;
END_VAR
VAR_OUTPUT
    VO_Drift_Detected : BOOL;
    VO_Drift_Score : UINT;

    VO_Status_Code : UINT;
    VO_Status_Text : STRING(128);
END_VAR
VAR
    L_Delta : UINT;
END_VAR

VO_Drift_Detected := FALSE;
VO_Drift_Score := 0;

VO_Status_Code := 0;
VO_Status_Text := 'Heating adaptive drift detector disabled';

IF NOT VI_Enable THEN
    RETURN;
END_IF;

IF VI_Runtime_Risk > VI_Runtime_Stability THEN
    L_Delta := VI_Runtime_Risk - VI_Runtime_Stability;
ELSE
    L_Delta := VI_Runtime_Stability - VI_Runtime_Risk;
END_IF;

VO_Drift_Score := L_Delta;
VO_Drift_Detected := (L_Delta > 40);

IF VO_Drift_Detected THEN
    VO_Status_Code := 200;
    VO_Status_Text := 'Heating adaptive supervision drift detected';
ELSE
    VO_Status_Code := 1;
    VO_Status_Text := 'Heating adaptive supervision stable';
END_IF;

END_FUNCTION_BLOCK
// >>> BULK_SYNC_ANCHOR: FB_Heating_Runtime_Adaptive_Drift_Detector <<<

(* ---- FB_Heating_Runtime_Anomaly_Aggregator.st ---- *)
// ==============================================================================
// Heating runtime anomaly aggregator
// Read-only anomaly aggregation layer.
// ==============================================================================
FUNCTION_BLOCK FB_Heating_Runtime_Anomaly_Aggregator
VAR_INPUT
    VI_Enable : BOOL;
    VI_Anomaly : ST_Heating_Runtime_Anomaly;
    VI_OT_Cascade_Correlation : BOOL;
END_VAR
VAR_OUTPUT
    VO_Runtime_Degraded : BOOL;
    VO_Runtime_Critical : BOOL;

    VO_Status_Code : UINT;
    VO_Status_Text : STRING(128);
END_VAR

VO_Runtime_Degraded := FALSE;
VO_Runtime_Critical := FALSE;

VO_Status_Code := 0;
VO_Status_Text := 'Heating runtime anomaly aggregator disabled';

IF NOT VI_Enable THEN
    RETURN;
END_IF;

IF VI_Anomaly.Critical_Anomaly THEN
    VO_Runtime_Critical := TRUE;

    VO_Status_Code := 900;
    VO_Status_Text := 'Heating runtime critical anomaly';

ELSIF VI_Anomaly.Anomaly_Active OR
      VI_OT_Cascade_Correlation THEN

    VO_Runtime_Degraded := TRUE;

    VO_Status_Code := 200;
    VO_Status_Text := 'Heating runtime degraded anomaly state';

ELSE
    VO_Status_Code := 1;
    VO_Status_Text := 'Heating runtime anomaly nominal';
END_IF;

END_FUNCTION_BLOCK
// >>> BULK_SYNC_ANCHOR: FB_Heating_Runtime_Anomaly_Aggregator <<<

(* ---- FB_Heating_Runtime_Anomaly_Weighting_Engine.st ---- *)
// ==============================================================================
// Heating runtime anomaly weighting engine
// Read-only adaptive anomaly weighting layer.
// ==============================================================================
FUNCTION_BLOCK FB_Heating_Runtime_Anomaly_Weighting_Engine
VAR_INPUT
    VI_Enable : BOOL;
    VI_Runtime_Degraded : BOOL;
    VI_Cascade_Degraded : BOOL;
    VI_OT_Degraded : BOOL;
    VI_Diagnostics_Degraded : BOOL;
END_VAR
VAR_OUTPUT
    VO_Runtime_Weight : UINT;
    VO_Cascade_Weight : UINT;
    VO_OT_Weight : UINT;
    VO_Diagnostics_Weight : UINT;

    VO_Status_Code : UINT;
    VO_Status_Text : STRING(128);
END_VAR

VO_Runtime_Weight := 0;
VO_Cascade_Weight := 0;
VO_OT_Weight := 0;
VO_Diagnostics_Weight := 0;

VO_Status_Code := 0;
VO_Status_Text := 'Heating anomaly weighting engine disabled';

IF NOT VI_Enable THEN
    RETURN;
END_IF;

IF VI_Runtime_Degraded THEN
    VO_Runtime_Weight := 80;
ELSE
    VO_Runtime_Weight := 10;
END_IF;

IF VI_Cascade_Degraded THEN
    VO_Cascade_Weight := 70;
ELSE
    VO_Cascade_Weight := 10;
END_IF;

IF VI_OT_Degraded THEN
    VO_OT_Weight := 75;
ELSE
    VO_OT_Weight := 10;
END_IF;

IF VI_Diagnostics_Degraded THEN
    VO_Diagnostics_Weight := 40;
ELSE
    VO_Diagnostics_Weight := 5;
END_IF;

VO_Status_Code := 1;
VO_Status_Text := 'Heating anomaly weighting updated';

END_FUNCTION_BLOCK
// >>> BULK_SYNC_ANCHOR: FB_Heating_Runtime_Anomaly_Weighting_Engine <<<

(* ---- FB_Heating_Runtime_Cascade_Collapse_Predictor.st ---- *)
// ==============================================================================
// Heating runtime cascade collapse predictor
// Read-only predictive cascade supervision layer.
// ==============================================================================
FUNCTION_BLOCK FB_Heating_Runtime_Cascade_Collapse_Predictor
VAR_INPUT
    VI_Enable : BOOL;
    VI_Cascade_Degraded : BOOL;
    VI_Active_Boilers : UINT;
END_VAR
VAR_OUTPUT
    VO_Cascade_Collapse_Risk : UINT;
    VO_Cascade_Degraded_Trend : BOOL;

    VO_Status_Code : UINT;
    VO_Status_Text : STRING(128);
END_VAR

VO_Cascade_Collapse_Risk := 0;
VO_Cascade_Degraded_Trend := FALSE;

VO_Status_Code := 0;
VO_Status_Text := 'Heating runtime cascade predictor disabled';

IF NOT VI_Enable THEN
    RETURN;
END_IF;

IF (VI_Active_Boilers = 0) THEN
    VO_Cascade_Collapse_Risk := 100;
    VO_Cascade_Degraded_Trend := TRUE;

    VO_Status_Code := 900;
    VO_Status_Text := 'Heating runtime cascade collapse predicted';

ELSIF VI_Cascade_Degraded THEN
    VO_Cascade_Collapse_Risk := 60;
    VO_Cascade_Degraded_Trend := TRUE;

    VO_Status_Code := 200;
    VO_Status_Text := 'Heating runtime cascade degradation trend';

ELSE
    VO_Cascade_Collapse_Risk := 5;

    VO_Status_Code := 1;
    VO_Status_Text := 'Heating runtime cascade nominal';
END_IF;

END_FUNCTION_BLOCK
// >>> BULK_SYNC_ANCHOR: FB_Heating_Runtime_Cascade_Collapse_Predictor <<<

(* ---- FB_Heating_Runtime_Causality_Propagation_Analyzer.st ---- *)
// ==============================================================================
// Heating runtime causality propagation analyzer
// Read-only runtime propagation analysis layer.
// ==============================================================================
FUNCTION_BLOCK FB_Heating_Runtime_Causality_Propagation_Analyzer
VAR_INPUT
    VI_Enable : BOOL;
    VI_Node : ST_Heating_Runtime_Causality_Node;
END_VAR
VAR_OUTPUT
    VO_Edge : ST_Heating_Runtime_Causality_Edge;
END_VAR

VO_Edge.Edge_Active := FALSE;
VO_Edge.Propagation_Detected := FALSE;

VO_Edge.Status_Code := 0;
VO_Edge.Status_Text := 'Heating runtime causality propagation analyzer disabled';

IF NOT VI_Enable THEN
    RETURN;
END_IF;

VO_Edge.Edge_Active := VI_Node.Node_Active;

VO_Edge.Runtime_Propagation :=
    VI_Node.Runtime_Degraded;

VO_Edge.Cascade_Propagation :=
    VI_Node.Cascade_Degraded OR
    VI_Node.Cascade_Boiler_Loss;

VO_Edge.OpenTherm_Propagation :=
    VI_Node.OpenTherm_Degraded OR
    VI_Node.OpenTherm_Command_Invalid;

VO_Edge.Diagnostics_Propagation :=
    VI_Node.Diagnostics_Degraded OR
    VI_Node.Explainability_Degraded;

VO_Edge.Sequencing_Propagation :=
    VI_Node.Sequencing_Invalid;

VO_Edge.Ownership_Propagation :=
    VI_Node.Ownership_Invalid;

VO_Edge.Synchronization_Propagation :=
    VI_Node.Synchronization_Invalid;

VO_Edge.Propagation_Detected :=
    VO_Edge.Runtime_Propagation OR
    VO_Edge.Cascade_Propagation OR
    VO_Edge.OpenTherm_Propagation OR
    VO_Edge.Diagnostics_Propagation OR
    VO_Edge.Sequencing_Propagation OR
    VO_Edge.Ownership_Propagation OR
    VO_Edge.Synchronization_Propagation;

VO_Edge.Severity_Level := VI_Node.Severity_Level;

VO_Edge.Critical_Path :=
    VI_Node.Root_Cause_Candidate;

IF VO_Edge.Critical_Path THEN
    VO_Edge.Status_Code := 900;
    VO_Edge.Status_Text := 'Heating runtime critical propagation path';
ELSIF VO_Edge.Propagation_Detected THEN
    VO_Edge.Status_Code := 200;
    VO_Edge.Status_Text := 'Heating runtime propagation detected';
ELSE
    VO_Edge.Status_Code := 1;
    VO_Edge.Status_Text := 'Heating runtime propagation nominal';
END_IF;

END_FUNCTION_BLOCK
// >>> BULK_SYNC_ANCHOR: FB_Heating_Runtime_Causality_Propagation_Analyzer <<<

(* ---- FB_Heating_Runtime_Coordinator.st ---- *)
// ==============================================================================
// Heating runtime coordinator
// Safe orchestration shell.
// DOES NOT own heating logic.
// DOES NOT own diagnostics.
// DOES NOT own OpenTherm transport.
// DOES NOT own safety.
// ==============================================================================
FUNCTION_BLOCK FB_Heating_Runtime_Coordinator
VAR_INPUT
    VI_Enable : BOOL;
END_VAR
VAR_OUTPUT
    // Typed runtime context
    VO_Runtime_Context : ST_Heating_Runtime_Context;

    // Current runtime phase
    VO_Current_Phase : E_Heating_Runtime_Phase;

    // Phase execution flags
    VO_Run_DHW_Phase : BOOL;
    VO_Run_Heating_Phase : BOOL;
    VO_Run_Service_Gating_Phase : BOOL;
    VO_Run_State_Publication_Phase : BOOL;
    VO_Run_Diagnostics_Phase : BOOL;
    VO_Run_Output_Projection_Phase : BOOL;

    // Runtime state
    VO_Runtime_Ready : BOOL;
    VO_Runtime_Fault : BOOL;
    VO_Runtime_Status_Text : STRING(128);
END_VAR
VAR
    L_Runtime_Valid : BOOL;
END_VAR

// ======================================================
// DEFAULTS
// ======================================================
VO_Runtime_Context.Runtime_Enabled := FALSE;
VO_Runtime_Context.Runtime_Ready := FALSE;
VO_Runtime_Context.Runtime_Fault := FALSE;
VO_Runtime_Context.Current_Phase := E_Heating_Runtime_Phase.HRP_DISABLED;

VO_Runtime_Context.Allow_DHW_Phase := FALSE;
VO_Runtime_Context.Allow_Heating_Phase := FALSE;
VO_Runtime_Context.Allow_Service_Gating_Phase := FALSE;
VO_Runtime_Context.Allow_State_Publication_Phase := FALSE;
VO_Runtime_Context.Allow_Diagnostics_Phase := FALSE;
VO_Runtime_Context.Allow_Output_Projection_Phase := FALSE;

VO_Runtime_Context.DHW_Executed := FALSE;
VO_Runtime_Context.Heating_Executed := FALSE;
VO_Runtime_Context.Service_Gating_Executed := FALSE;
VO_Runtime_Context.State_Publication_Executed := FALSE;
VO_Runtime_Context.Diagnostics_Executed := FALSE;
VO_Runtime_Context.Output_Projection_Executed := FALSE;

VO_Runtime_Context.DHW_Before_Heating_Valid := TRUE;
VO_Runtime_Context.State_Publication_Before_Diagnostics_Valid := TRUE;
VO_Runtime_Context.Output_Projection_Last_Valid := TRUE;

VO_Runtime_Context.Diagnostics_Isolation_Valid := TRUE;
VO_Runtime_Context.Explainability_Isolation_Valid := TRUE;
VO_Runtime_Context.Safety_Isolation_Valid := TRUE;
VO_Runtime_Context.OpenTherm_Ownership_Valid := TRUE;
VO_Runtime_Context.Cascade_Ownership_Valid := TRUE;

VO_Runtime_Context.Runtime_Status_Code := 0;
VO_Runtime_Context.Runtime_Status_Text := 'Heating runtime coordinator disabled';

VO_Current_Phase := E_Heating_Runtime_Phase.HRP_DISABLED;

VO_Run_DHW_Phase := FALSE;
VO_Run_Heating_Phase := FALSE;
VO_Run_Service_Gating_Phase := FALSE;
VO_Run_State_Publication_Phase := FALSE;
VO_Run_Diagnostics_Phase := FALSE;
VO_Run_Output_Projection_Phase := FALSE;

VO_Runtime_Ready := FALSE;
VO_Runtime_Fault := FALSE;
VO_Runtime_Status_Text := 'Heating runtime coordinator disabled';

L_Runtime_Valid := FALSE;

IF NOT VI_Enable THEN
    RETURN;
END_IF;

// ======================================================
// RUNTIME CONTRACT VALIDATION
// ======================================================
L_Runtime_Valid := TRUE;

IF NOT L_Runtime_Valid THEN
    VO_Current_Phase := E_Heating_Runtime_Phase.HRP_FAULT;

    VO_Runtime_Context.Runtime_Enabled := TRUE;
    VO_Runtime_Context.Runtime_Ready := FALSE;
    VO_Runtime_Context.Runtime_Fault := TRUE;
    VO_Runtime_Context.Current_Phase := E_Heating_Runtime_Phase.HRP_FAULT;
    VO_Runtime_Context.Runtime_Status_Code := 900;
    VO_Runtime_Context.Runtime_Status_Text := 'Heating runtime sequencing invalid';

    VO_Runtime_Ready := FALSE;
    VO_Runtime_Fault := TRUE;
    VO_Runtime_Status_Text := 'Heating runtime sequencing invalid';
    RETURN;
END_IF;

// ======================================================
// PHASE 1 — DHW
// ======================================================
VO_Current_Phase := E_Heating_Runtime_Phase.HRP_DHW;
VO_Run_DHW_Phase := TRUE;

VO_Runtime_Context.Runtime_Enabled := TRUE;
VO_Runtime_Context.Allow_DHW_Phase := TRUE;
VO_Runtime_Context.Current_Phase := E_Heating_Runtime_Phase.HRP_DHW;
VO_Runtime_Context.DHW_Executed := TRUE;

// ======================================================
// PHASE 2 — HEATING
// ======================================================
VO_Current_Phase := E_Heating_Runtime_Phase.HRP_HEATING;
VO_Run_Heating_Phase := TRUE;

VO_Runtime_Context.Allow_Heating_Phase := TRUE;
VO_Runtime_Context.Current_Phase := E_Heating_Runtime_Phase.HRP_HEATING;
VO_Runtime_Context.Heating_Executed := TRUE;

// ======================================================
// PHASE 3 — SERVICE / FAILSAFE GATING
// ======================================================
VO_Current_Phase := E_Heating_Runtime_Phase.HRP_SERVICE_GATING;
VO_Run_Service_Gating_Phase := TRUE;

VO_Runtime_Context.Allow_Service_Gating_Phase := TRUE;
VO_Runtime_Context.Current_Phase := E_Heating_Runtime_Phase.HRP_SERVICE_GATING;
VO_Runtime_Context.Service_Gating_Executed := TRUE;

// ======================================================
// PHASE 4 — STATE PUBLICATION
// ======================================================
VO_Current_Phase := E_Heating_Runtime_Phase.HRP_STATE_PUBLICATION;
VO_Run_State_Publication_Phase := TRUE;

VO_Runtime_Context.Allow_State_Publication_Phase := TRUE;
VO_Runtime_Context.Current_Phase := E_Heating_Runtime_Phase.HRP_STATE_PUBLICATION;
VO_Runtime_Context.State_Publication_Executed := TRUE;

// ======================================================
// PHASE 5 — DIAGNOSTICS
// ======================================================
VO_Current_Phase := E_Heating_Runtime_Phase.HRP_DIAGNOSTICS;
VO_Run_Diagnostics_Phase := TRUE;

VO_Runtime_Context.Allow_Diagnostics_Phase := TRUE;
VO_Runtime_Context.Current_Phase := E_Heating_Runtime_Phase.HRP_DIAGNOSTICS;
VO_Runtime_Context.Diagnostics_Executed := TRUE;

// ======================================================
// PHASE 6 — OUTPUT PROJECTION
// ======================================================
VO_Current_Phase := E_Heating_Runtime_Phase.HRP_OUTPUT_PROJECTION;
VO_Run_Output_Projection_Phase := TRUE;

VO_Runtime_Context.Allow_Output_Projection_Phase := TRUE;
VO_Runtime_Context.Current_Phase := E_Heating_Runtime_Phase.HRP_OUTPUT_PROJECTION;
VO_Runtime_Context.Output_Projection_Executed := TRUE;

// ======================================================
// COMPLETE
// ======================================================
VO_Current_Phase := E_Heating_Runtime_Phase.HRP_COMPLETE;
VO_Runtime_Context.Current_Phase := E_Heating_Runtime_Phase.HRP_COMPLETE;

VO_Runtime_Context.Runtime_Ready := TRUE;
VO_Runtime_Context.Runtime_Fault := FALSE;
VO_Runtime_Context.Runtime_Status_Code := 100;
VO_Runtime_Context.Runtime_Status_Text := 'Heating runtime coordinator active';

VO_Runtime_Ready := TRUE;
VO_Runtime_Fault := FALSE;
VO_Runtime_Status_Text := 'Heating runtime coordinator active';

END_FUNCTION_BLOCK
// >>> BULK_SYNC_ANCHOR: FB_Heating_Runtime_Coordinator <<<

(* ---- FB_Heating_Runtime_Degradation_Timeline_Rebuilder.st ---- *)
// ==============================================================================
// Heating runtime degradation timeline rebuilder
// Read-only runtime degradation reconstruction layer.
// ==============================================================================
FUNCTION_BLOCK FB_Heating_Runtime_Degradation_Timeline_Rebuilder
VAR_INPUT
    VI_Enable : BOOL;
    VI_Event : ST_Heating_Runtime_Blackbox_Event;
END_VAR
VAR_IN_OUT
    VIO_Timeline : ST_Heating_Runtime_Blackbox_Timeline;
END_VAR
VAR
    L_Index : UINT;
END_VAR

IF NOT VI_Enable THEN
    RETURN;
END_IF;

// ======================================================
// SAFE INDEX NORMALIZATION
// ======================================================
IF (VIO_Timeline.Write_Index < 1) OR
   (VIO_Timeline.Write_Index >= 256) THEN

    L_Index := 1;

    IF VIO_Timeline.Write_Index >= 256 THEN
        VIO_Timeline.Timeline_Overflow := TRUE;
    END_IF;

ELSE
    L_Index := VIO_Timeline.Write_Index + 1;
END_IF;

// ======================================================
// EVENT STORAGE
// ======================================================
VIO_Timeline.Events[L_Index] := VI_Event;
VIO_Timeline.Write_Index := L_Index;

IF VIO_Timeline.Event_Count < 256 THEN
    VIO_Timeline.Event_Count :=
        VIO_Timeline.Event_Count + 1;
END_IF;

// ======================================================
// TIMELINE STATE UPDATE
// ======================================================
VIO_Timeline.Reconstruction_Active := TRUE;
VIO_Timeline.Replay_Active := VI_Event.Event_Active;

VIO_Timeline.Root_Cause_Reconstructed :=
    VI_Event.Root_Cause_Candidate;

VIO_Timeline.Sequencing_Valid :=
    NOT VI_Event.Sequencing_Invalid;

VIO_Timeline.Ownership_Valid :=
    NOT VI_Event.Ownership_Invalid;

VIO_Timeline.Synchronization_Valid :=
    NOT VI_Event.Synchronization_Invalid;

IF VI_Event.Root_Cause_Candidate THEN
    VIO_Timeline.Status_Code := 900;
    VIO_Timeline.Status_Text := 'Heating runtime degradation reconstructed';
ELSE
    VIO_Timeline.Status_Code := 1;
    VIO_Timeline.Status_Text := 'Heating runtime forensic timeline nominal';
END_IF;

END_FUNCTION_BLOCK
// >>> BULK_SYNC_ANCHOR: FB_Heating_Runtime_Degradation_Timeline_Rebuilder <<<

(* ---- FB_Heating_Runtime_Degradation_Trend_Analyzer.st ---- *)
// ==============================================================================
// Heating runtime degradation trend analyzer
// Read-only predictive degradation trend layer.
// ==============================================================================
FUNCTION_BLOCK FB_Heating_Runtime_Degradation_Trend_Analyzer
VAR_INPUT
    VI_Enable : BOOL;
    VI_Runtime_Degraded : BOOL;
    VI_Runtime_Critical : BOOL;
END_VAR
VAR_OUTPUT
    VO_Degradation_Risk : UINT;
    VO_Failure_Probability : UINT;

    VO_Status_Code : UINT;
    VO_Status_Text : STRING(128);
END_VAR

VO_Degradation_Risk := 0;
VO_Failure_Probability := 0;

VO_Status_Code := 0;
VO_Status_Text := 'Heating runtime degradation trend analyzer disabled';

IF NOT VI_Enable THEN
    RETURN;
END_IF;

IF VI_Runtime_Critical THEN
    VO_Degradation_Risk := 100;
    VO_Failure_Probability := 95;

    VO_Status_Code := 900;
    VO_Status_Text := 'Heating runtime failure risk critical';

ELSIF VI_Runtime_Degraded THEN
    VO_Degradation_Risk := 60;
    VO_Failure_Probability := 40;

    VO_Status_Code := 200;
    VO_Status_Text := 'Heating runtime degradation trend detected';

ELSE
    VO_Degradation_Risk := 10;
    VO_Failure_Probability := 5;

    VO_Status_Code := 1;
    VO_Status_Text := 'Heating runtime degradation nominal';
END_IF;

END_FUNCTION_BLOCK
// >>> BULK_SYNC_ANCHOR: FB_Heating_Runtime_Degradation_Trend_Analyzer <<<

(* ---- FB_Heating_Runtime_Event_Reconstruction_Engine.st ---- *)
// ==============================================================================
// Heating runtime event reconstruction engine
// Read-only runtime forensic reconstruction layer.
// ==============================================================================
FUNCTION_BLOCK FB_Heating_Runtime_Event_Reconstruction_Engine
VAR_INPUT
    VI_Enable : BOOL;
    VI_Node : ST_Heating_Runtime_Causality_Node;
    VI_Edge : ST_Heating_Runtime_Causality_Edge;
    VI_System_Time_MS : UDINT;
END_VAR
VAR_OUTPUT
    VO_Event : ST_Heating_Runtime_Blackbox_Event;
END_VAR

VO_Event.Event_Active := FALSE;
VO_Event.Root_Cause_Candidate := FALSE;
VO_Event.Critical_Path := FALSE;

VO_Event.Status_Code := 0;
VO_Event.Status_Text := 'Heating runtime reconstruction engine disabled';

IF NOT VI_Enable THEN
    RETURN;
END_IF;

VO_Event.Event_Active := VI_Node.Node_Active;
VO_Event.Runtime_Phase := E_Heating_Runtime_Phase.HRP_COMPLETE;

VO_Event.Event_Start_MS := VI_System_Time_MS;
VO_Event.Event_End_MS := VI_System_Time_MS;
VO_Event.Event_Duration_MS := 0;

VO_Event.Runtime_Degraded := VI_Node.Runtime_Degraded;
VO_Event.Runtime_Fault := VI_Node.Runtime_Fault;

VO_Event.Cascade_Degraded := VI_Node.Cascade_Degraded;
VO_Event.Cascade_Boiler_Loss := VI_Node.Cascade_Boiler_Loss;

VO_Event.OpenTherm_Degraded := VI_Node.OpenTherm_Degraded;
VO_Event.OpenTherm_Command_Invalid :=
    VI_Node.OpenTherm_Command_Invalid;

VO_Event.Sequencing_Invalid :=
    VI_Node.Sequencing_Invalid;

VO_Event.Ownership_Invalid :=
    VI_Node.Ownership_Invalid;

VO_Event.Synchronization_Invalid :=
    VI_Node.Synchronization_Invalid;

VO_Event.Root_Cause_Candidate :=
    VI_Node.Root_Cause_Candidate;

VO_Event.Critical_Path :=
    VI_Edge.Critical_Path;

IF VO_Event.Root_Cause_Candidate THEN
    VO_Event.Status_Code := 900;
    VO_Event.Status_Text := 'Heating runtime root-cause reconstructed';
ELSE
    VO_Event.Status_Code := 1;
    VO_Event.Status_Text := 'Heating runtime event reconstructed';
END_IF;

END_FUNCTION_BLOCK
// >>> BULK_SYNC_ANCHOR: FB_Heating_Runtime_Event_Reconstruction_Engine <<<
